   1:  PR[91,1] = PR[90,1] + 29.566;
   1:  PR[91,2] = PR[90,2] + 8.406;
   1:L PR[91] R[100]mm/sec CNT100;
   1:  PR[91,1] = PR[90,1] + 27.904;
   1:  PR[91,2] = PR[90,2] + 11.117;
   1:L PR[91] R[100]mm/sec CNT100;
   1:  PR[91,1] = PR[90,1] + 27.115;
   1:  PR[91,2] = PR[90,2] + 12.361;
   1:L PR[91] R[100]mm/sec CNT100;
   1:  PR[91,1] = PR[90,1] + 24.735;
   1:  PR[91,2] = PR[90,2] + 14.832;
   1:L PR[91] R[100]mm/sec CNT100;
   1:  PR[91,1] = PR[90,1] + 23.842;
   1:  PR[91,2] = PR[90,2] + 15.724;
   1:L PR[91] R[100]mm/sec CNT100;
   1:  PR[91,1] = PR[90,1] + 20.728;
   1:  PR[91,2] = PR[90,2] + 17.807;
   1:L PR[91] R[100]mm/sec CNT100;
   1:  PR[91,1] = PR[90,1] + 19.885;
   1:  PR[91,2] = PR[90,2] + 18.343;
   1:L PR[91] R[100]mm/sec CNT100;
   1:  PR[91,1] = PR[90,1] + 16.075;
   1:  PR[91,2] = PR[90,2] + 19.861;
   1:L PR[91] R[100]mm/sec CNT100;
   1:  PR[91,1] = PR[90,1] + 15.423;
   1:  PR[91,2] = PR[90,2] + 20.103;
   1:L PR[91] R[100]mm/sec CNT100;
   1:  PR[91,1] = PR[90,1] + 11.037;
   1:  PR[91,2] = PR[90,2] + 20.852;
   1:L PR[91] R[100]mm/sec CNT100;
   1:  PR[91,1] = PR[90,1] + 10.671;
   1:  PR[91,2] = PR[90,2] + 20.905;
   1:L PR[91] R[100]mm/sec CNT100;
   1:  PR[91,1] = PR[90,1] + 5.819;
   1:  PR[91,2] = PR[90,2] + 20.698;
   1:L PR[91] R[100]mm/sec CNT100;
   1:  PR[91,1] = PR[90,1] + 2.434;
   1:  PR[91,2] = PR[90,2] + 19.809;
   1:L PR[91] R[100]mm/sec CNT100;
   1:  PR[91,1] = PR[90,1] + 1.059;
   1:  PR[91,2] = PR[90,2] + 19.465;
   1:L PR[91] R[100]mm/sec CNT100;
   1:  PR[91,1] = PR[90,1] + 0.436;
   1:  PR[91,2] = PR[90,2] + 19.230;
   1:L PR[91] R[100]mm/sec CNT100;
   1:  PR[91] = PR[90];
   1:  PR[91,1] = PR[90,1] + -0.654;
   1:  PR[91,2] = PR[90,2] + 19.657;
   1:  PR[91,3] = PR[90,3] + 50.895;
   1:L PR[91] R[100]mm/sec CNT100;
   1:  PR[91,1] = PR[90,1] + -1.326;
   1:  PR[91,2] = PR[90,2] + 19.800;
   1:L PR[91] R[100]mm/sec CNT100;
   1:  PR[91,1] = PR[90,1] + -5.785;
   1:  PR[91,2] = PR[90,2] + 20.909;
   1:L PR[91] R[100]mm/sec CNT100;
   1:  PR[91,1] = PR[90,1] + -10.696;
   1:  PR[91,2] = PR[90,2] + 21.085;
   1:L PR[91] R[100]mm/sec CNT100;
   1:  PR[91,1] = PR[90,1] + -15.480;
   1:  PR[91,2] = PR[90,2] + 20.269;
   1:L PR[91] R[100]mm/sec CNT100;
   1:  PR[91,1] = PR[90,1] + -19.985;
   1:  PR[91,2] = PR[90,2] + 18.481;
   1:L PR[91] R[100]mm/sec CNT100;
   1:  PR[91,1] = PR[90,1] + -20.308;
   1:  PR[91,2] = PR[90,2] + 18.276;
   1:L PR[91] R[100]mm/sec CNT100;
   1:  PR[91,1] = PR[90,1] + -23.955;
   1:  PR[91,2] = PR[90,2] + 15.836;
   1:L PR[91] R[100]mm/sec CNT100;
   1:  PR[91,1] = PR[90,1] + -24.411;
   1:  PR[91,2] = PR[90,2] + 15.381;
   1:L PR[91] R[100]mm/sec CNT100;
   1:  PR[91,1] = PR[90,1] + -27.236;
   1:  PR[91,2] = PR[90,2] + 12.453;
   1:L PR[91] R[100]mm/sec CNT100;
   1:  PR[91,1] = PR[90,1] + -27.694;
   1:  PR[91,2] = PR[90,2] + 11.729;
   1:L PR[91] R[100]mm/sec CNT100;
   1:  PR[91,1] = PR[90,1] + -29.692;
   1:  PR[91,2] = PR[90,2] + 8.469;
   1:L PR[91] R[100]mm/sec CNT100;
   1:  PR[91,1] = PR[90,1] + -30.028;
   1:  PR[91,2] = PR[90,2] + 7.542;
   1:L PR[91] R[100]mm/sec CNT100;
   1:  PR[91,1] = PR[90,1] + -31.203;
   1:  PR[91,2] = PR[90,2] + 4.166;
   1:L PR[91] R[100]mm/sec CNT100;
   1:  PR[91,1] = PR[90,1] + -31.322;
   1:  PR[91,2] = PR[90,2] + 3.118;
   1:L PR[91] R[100]mm/sec CNT100;
   1:  PR[91,1] = PR[90,1] + -31.390;
   1:  PR[91,2] = PR[90,2] + 2.274;
   1:L PR[91] R[100]mm/sec CNT100;
   1:  PR[91,1] = PR[90,1] + -31.692;
   1:  PR[91,2] = PR[90,2] + -0.443;
   1:L PR[91] R[100]mm/sec CNT100;
   1:  PR[91,1] = PR[90,1] + -31.586;
   1:  PR[91,2] = PR[90,2] + -1.550;
   1:L PR[91] R[100]mm/sec CNT100;
   1:  PR[91,1] = PR[90,1] + -31.201;
   1:  PR[91,2] = PR[90,2] + -5.016;
   1:L PR[91] R[100]mm/sec CNT100;
   1:  PR[91,1] = PR[90,1] + -30.028;
   1:  PR[91,2] = PR[90,2] + -8.389;
   1:L PR[91] R[100]mm/sec CNT100;
   1:  PR[91,1] = PR[90,1] + -29.692;
   1:  PR[91,2] = PR[90,2] + -9.316;
   1:L PR[91] R[100]mm/sec CNT100;
   1:  PR[91,1] = PR[90,1] + -27.694;
   1:  PR[91,2] = PR[90,2] + -12.577;
   1:L PR[91] R[100]mm/sec CNT100;
   1:  PR[91,1] = PR[90,1] + -27.236;
   1:  PR[91,2] = PR[90,2] + -13.301;
   1:L PR[91] R[100]mm/sec CNT100;
   1:  PR[91,1] = PR[90,1] + -24.411;
   1:  PR[91,2] = PR[90,2] + -16.228;
   1:L PR[91] R[100]mm/sec CNT100;
   1:  PR[91,1] = PR[90,1] + -23.955;
   1:  PR[91,2] = PR[90,2] + -16.683;
   1:L PR[91] R[100]mm/sec CNT100;
   1:  PR[91,1] = PR[90,1] + -20.307;
   1:  PR[91,2] = PR[90,2] + -19.123;
   1:L PR[91] R[100]mm/sec CNT100;
   1:  PR[91,1] = PR[90,1] + -19.985;
   1:  PR[91,2] = PR[90,2] + -19.329;
   1:L PR[91] R[100]mm/sec CNT100;
   1:  PR[91,1] = PR[90,1] + -15.480;
   1:  PR[91,2] = PR[90,2] + -21.116;
   1:L PR[91] R[100]mm/sec CNT100;
   1:  PR[91,1] = PR[90,1] + -10.696;
   1:  PR[91,2] = PR[90,2] + -21.933;
   1:L PR[91] R[100]mm/sec CNT100;
   1:  PR[91,1] = PR[90,1] + -5.784;
   1:  PR[91,2] = PR[90,2] + -21.756;
   1:L PR[91] R[100]mm/sec CNT100;
   1:  PR[91,1] = PR[90,1] + -1.093;
   1:  PR[91,2] = PR[90,2] + -20.590;
   1:L PR[91] R[100]mm/sec CNT100;
   1:  PR[91,1] = PR[90,1] + -0.762;
   1:  PR[91,2] = PR[90,2] + -20.587;
   1:L PR[91] R[100]mm/sec CNT100;
   1:  PR[91,1] = PR[90,1] + 0.330;
   1:  PR[91,2] = PR[90,2] + -20.423;
   1:L PR[91] R[100]mm/sec CNT100;
   1:  PR[91,1] = PR[90,1] + 1.032;
   1:  PR[91,2] = PR[90,2] + -20.694;
   1:L PR[91] R[100]mm/sec CNT100;
   1:  PR[91,1] = PR[90,1] + 5.305;
   1:  PR[91,2] = PR[90,2] + -21.756;
   1:L PR[91] R[100]mm/sec CNT100;
   1:  PR[91,1] = PR[90,1] + 10.217;
   1:  PR[91,2] = PR[90,2] + -21.933;
   1:L PR[91] R[100]mm/sec CNT100;
   1:  PR[91,1] = PR[90,1] + 15.000;
   1:  PR[91,2] = PR[90,2] + -21.116;
   1:L PR[91] R[100]mm/sec CNT100;
   1:  PR[91,1] = PR[90,1] + 19.507;
   1:  PR[91,2] = PR[90,2] + -19.329;
   1:L PR[91] R[100]mm/sec CNT100;
   1:  PR[91,1] = PR[90,1] + 19.829;
   1:  PR[91,2] = PR[90,2] + -19.124;
   1:L PR[91] R[100]mm/sec CNT100;
   1:  PR[91,1] = PR[90,1] + 23.474;
   1:  PR[91,2] = PR[90,2] + -16.686;
   1:L PR[91] R[100]mm/sec CNT100;
   1:  PR[91,1] = PR[90,1] + 23.930;
   1:  PR[91,2] = PR[90,2] + -16.231;
   1:L PR[91] R[100]mm/sec CNT100;
   1:  PR[91,1] = PR[90,1] + 26.756;
   1:  PR[91,2] = PR[90,2] + -13.296;
   1:L PR[91] R[100]mm/sec CNT100;
   1:  PR[91,1] = PR[90,1] + 27.215;
   1:  PR[91,2] = PR[90,2] + -12.572;
   1:L PR[91] R[100]mm/sec CNT100;
   1:  PR[91,1] = PR[90,1] + 29.213;
   1:  PR[91,2] = PR[90,2] + -9.314;
   1:L PR[91] R[100]mm/sec CNT100;
   1:  PR[91,1] = PR[90,1] + 29.549;
   1:  PR[91,2] = PR[90,2] + -8.392;
   1:L PR[91] R[100]mm/sec CNT100;
   1:  PR[91,1] = PR[90,1] + 30.723;
   1:  PR[91,2] = PR[90,2] + -5.026;
   1:L PR[91] R[100]mm/sec CNT100;
   1:  PR[91,1] = PR[90,1] + 30.842;
   1:  PR[91,2] = PR[90,2] + -3.974;
   1:L PR[91] R[100]mm/sec CNT100;
   1:  PR[91,1] = PR[90,1] + 30.910;
   1:  PR[91,2] = PR[90,2] + -3.128;
   1:L PR[91] R[100]mm/sec CNT100;
   1:  PR[91,1] = PR[90,1] + 31.212;
   1:  PR[91,2] = PR[90,2] + -0.404;
   1:L PR[91] R[100]mm/sec CNT100;
   1:  PR[91,1] = PR[90,1] + 31.107;
   1:  PR[91,2] = PR[90,2] + 0.709;
   1:L PR[91] R[100]mm/sec CNT100;
   1:  PR[91,1] = PR[90,1] + 30.722;
   1:  PR[91,2] = PR[90,2] + 4.181;
   1:L PR[91] R[100]mm/sec CNT100;
   1:  PR[91,1] = PR[90,1] + 29.549;
   1:  PR[91,2] = PR[90,2] + 7.544;
   1:L PR[91] R[100]mm/sec CNT100;
   1:  PR[91,1] = PR[90,1] + 29.213;
   1:  PR[91,2] = PR[90,2] + 8.467;
   1:L PR[91] R[100]mm/sec CNT100;
   1:  PR[91,1] = PR[90,1] + 27.215;
   1:  PR[91,2] = PR[90,2] + 11.725;
   1:L PR[91] R[100]mm/sec CNT100;
   1:  PR[91,1] = PR[90,1] + 26.756;
   1:  PR[91,2] = PR[90,2] + 12.448;
   1:L PR[91] R[100]mm/sec CNT100;
   1:  PR[91,1] = PR[90,1] + 23.930;
   1:  PR[91,2] = PR[90,2] + 15.383;
   1:L PR[91] R[100]mm/sec CNT100;
   1:  PR[91,1] = PR[90,1] + 23.474;
   1:  PR[91,2] = PR[90,2] + 15.839;
   1:L PR[91] R[100]mm/sec CNT100;
   1:  PR[91,1] = PR[90,1] + 19.828;
   1:  PR[91,2] = PR[90,2] + 18.276;
   1:L PR[91] R[100]mm/sec CNT100;
   1:  PR[91,1] = PR[90,1] + 19.507;
   1:  PR[91,2] = PR[90,2] + 18.481;
   1:L PR[91] R[100]mm/sec CNT100;
   1:  PR[91,1] = PR[90,1] + 15.000;
   1:  PR[91,2] = PR[90,2] + 20.268;
   1:L PR[91] R[100]mm/sec CNT100;
   1:  PR[91,1] = PR[90,1] + 10.217;
   1:  PR[91,2] = PR[90,2] + 21.086;
   1:L PR[91] R[100]mm/sec CNT100;
   1:  PR[91,1] = PR[90,1] + 5.306;
   1:  PR[91,2] = PR[90,2] + 20.909;
   1:L PR[91] R[100]mm/sec CNT100;
   1:  PR[91,1] = PR[90,1] + 1.030;
   1:  PR[91,2] = PR[90,2] + 19.845;
   1:L PR[91] R[100]mm/sec CNT100;
   1:  PR[91,1] = PR[90,1] + 0.478;
   1:  PR[91,2] = PR[90,2] + 19.634;
   1:L PR[91] R[100]mm/sec CNT100;
   1:  PR[91] = PR[90];
   1:  PR[91,1] = PR[90,1] + -0.748;
   1:  PR[91,2] = PR[90,2] + 20.064;
   1:  PR[91,3] = PR[90,3] + 52.195;
   1:L PR[91] R[100]mm/sec CNT100;
   1:  PR[91,1] = PR[90,1] + -1.294;
   1:  PR[91,2] = PR[90,2] + 20.180;
   1:L PR[91] R[100]mm/sec CNT100;
   1:  PR[91,1] = PR[90,1] + -4.263;
   1:  PR[91,2] = PR[90,2] + 20.923;
   1:L PR[91] R[100]mm/sec CNT100;
   1:  PR[91,1] = PR[90,1] + -5.232;
   1:  PR[91,2] = PR[90,2] + 21.146;
   1:L PR[91] R[100]mm/sec CNT100;
   1:  PR[91,1] = PR[90,1] + -5.868;
   1:  PR[91,2] = PR[90,2] + 21.178;
   1:L PR[91] R[100]mm/sec CNT100;
   1:  PR[91,1] = PR[90,1] + -10.179;
   1:  PR[91,2] = PR[90,2] + 21.327;
   1:L PR[91] R[100]mm/sec CNT100;
   1:  PR[91,1] = PR[90,1] + -15.038;
   1:  PR[91,2] = PR[90,2] + 20.471;
   1:L PR[91] R[100]mm/sec CNT100;
   1:  PR[91,1] = PR[90,1] + -19.573;
   1:  PR[91,2] = PR[90,2] + 18.635;
   1:L PR[91] R[100]mm/sec CNT100;
   1:  PR[91,1] = PR[90,1] + -23.568;
   1:  PR[91,2] = PR[90,2] + 15.963;
   1:L PR[91] R[100]mm/sec CNT100;
   1:  PR[91,1] = PR[90,1] + -26.867;
   1:  PR[91,2] = PR[90,2] + 12.551;
   1:L PR[91] R[100]mm/sec CNT100;
   1:  PR[91,1] = PR[90,1] + -29.333;
   1:  PR[91,2] = PR[90,2] + 8.539;
   1:L PR[91] R[100]mm/sec CNT100;
   1:  PR[91,1] = PR[90,1] + -30.851;
   1:  PR[91,2] = PR[90,2] + 4.198;
   1:L PR[91] R[100]mm/sec CNT100;
   1:  PR[91,1] = PR[90,1] + -31.355;
   1:  PR[91,2] = PR[90,2] + -0.440;
   1:L PR[91] R[100]mm/sec CNT100;
   1:  PR[91,1] = PR[90,1] + -31.305;
   1:  PR[91,2] = PR[90,2] + -0.964;
   1:L PR[91] R[100]mm/sec CNT100;
   1:  PR[91,1] = PR[90,1] + -30.852;
   1:  PR[91,2] = PR[90,2] + -5.044;
   1:L PR[91] R[100]mm/sec CNT100;
   1:  PR[91,1] = PR[90,1] + -29.471;
   1:  PR[91,2] = PR[90,2] + -9.013;
   1:L PR[91] R[100]mm/sec CNT100;
   1:  PR[91,1] = PR[90,1] + -29.340;
   1:  PR[91,2] = PR[90,2] + -9.375;
   1:L PR[91] R[100]mm/sec CNT100;
   1:  PR[91,1] = PR[90,1] + -26.867;
   1:  PR[91,2] = PR[90,2] + -13.398;
   1:L PR[91] R[100]mm/sec CNT100;
   1:  PR[91,1] = PR[90,1] + -23.568;
   1:  PR[91,2] = PR[90,2] + -16.810;
   1:L PR[91] R[100]mm/sec CNT100;
   1:  PR[91,1] = PR[90,1] + -19.573;
   1:  PR[91,2] = PR[90,2] + -19.483;
   1:L PR[91] R[100]mm/sec CNT100;
   1:  PR[91,1] = PR[90,1] + -15.038;
   1:  PR[91,2] = PR[90,2] + -21.319;
   1:L PR[91] R[100]mm/sec CNT100;
   1:  PR[91,1] = PR[90,1] + -10.179;
   1:  PR[91,2] = PR[90,2] + -22.174;
   1:L PR[91] R[100]mm/sec CNT100;
   1:  PR[91,1] = PR[90,1] + -5.868;
   1:  PR[91,2] = PR[90,2] + -22.025;
   1:L PR[91] R[100]mm/sec CNT100;
   1:  PR[91,1] = PR[90,1] + -5.232;
   1:  PR[91,2] = PR[90,2] + -21.993;
   1:L PR[91] R[100]mm/sec CNT100;
   1:  PR[91,1] = PR[90,1] + -4.168;
   1:  PR[91,2] = PR[90,2] + -21.747;
   1:L PR[91] R[100]mm/sec CNT100;
   1:  PR[91,1] = PR[90,1] + -1.061;
   1:  PR[91,2] = PR[90,2] + -20.970;
   1:L PR[91] R[100]mm/sec CNT100;
   1:  PR[91,1] = PR[90,1] + -0.555;
   1:  PR[91,2] = PR[90,2] + -20.965;
   1:L PR[91] R[100]mm/sec CNT100;
   1:  PR[91,1] = PR[90,1] + 0.380;
   1:  PR[91,2] = PR[90,2] + -20.825;
   1:L PR[91] R[100]mm/sec CNT100;
   1:  PR[91,1] = PR[90,1] + 1.014;
   1:  PR[91,2] = PR[90,2] + -21.078;
   1:L PR[91] R[100]mm/sec CNT100;
   1:  PR[91,1] = PR[90,1] + 3.691;
   1:  PR[91,2] = PR[90,2] + -21.747;
   1:L PR[91] R[100]mm/sec CNT100;
   1:  PR[91,1] = PR[90,1] + 4.754;
   1:  PR[91,2] = PR[90,2] + -21.994;
   1:L PR[91] R[100]mm/sec CNT100;
   1:  PR[91,1] = PR[90,1] + 5.389;
   1:  PR[91,2] = PR[90,2] + -22.025;
   1:L PR[91] R[100]mm/sec CNT100;
   1:  PR[91,1] = PR[90,1] + 9.700;
   1:  PR[91,2] = PR[90,2] + -22.175;
   1:L PR[91] R[100]mm/sec CNT100;
   1:  PR[91,1] = PR[90,1] + 14.559;
   1:  PR[91,2] = PR[90,2] + -21.318;
   1:L PR[91] R[100]mm/sec CNT100;
   1:  PR[91,1] = PR[90,1] + 19.094;
   1:  PR[91,2] = PR[90,2] + -19.483;
   1:L PR[91] R[100]mm/sec CNT100;
   1:  PR[91,1] = PR[90,1] + 23.087;
   1:  PR[91,2] = PR[90,2] + -16.812;
   1:L PR[91] R[100]mm/sec CNT100;
   1:  PR[91,1] = PR[90,1] + 26.398;
   1:  PR[91,2] = PR[90,2] + -13.382;
   1:L PR[91] R[100]mm/sec CNT100;
   1:  PR[91,1] = PR[90,1] + 26.526;
   1:  PR[91,2] = PR[90,2] + -13.180;
   1:L PR[91] R[100]mm/sec CNT100;
   1:  PR[91,1] = PR[90,1] + 28.853;
   1:  PR[91,2] = PR[90,2] + -9.387;
   1:L PR[91] R[100]mm/sec CNT100;
   1:  PR[91,1] = PR[90,1] + 30.371;
   1:  PR[91,2] = PR[90,2] + -5.056;
   1:L PR[91] R[100]mm/sec CNT100;
   1:  PR[91,1] = PR[90,1] + 30.875;
   1:  PR[91,2] = PR[90,2] + -0.407;
   1:L PR[91] R[100]mm/sec CNT100;
   1:  PR[91,1] = PR[90,1] + 30.825;
   1:  PR[91,2] = PR[90,2] + 0.121;
   1:L PR[91] R[100]mm/sec CNT100;
   1:  PR[91,1] = PR[90,1] + 30.372;
   1:  PR[91,2] = PR[90,2] + 4.206;
   1:L PR[91] R[100]mm/sec CNT100;
   1:  PR[91,1] = PR[90,1] + 28.854;
   1:  PR[91,2] = PR[90,2] + 8.538;
   1:L PR[91] R[100]mm/sec CNT100;
   1:  PR[91,1] = PR[90,1] + 26.386;
   1:  PR[91,2] = PR[90,2] + 12.548;
   1:L PR[91] R[100]mm/sec CNT100;
   1:  PR[91,1] = PR[90,1] + 23.125;
   1:  PR[91,2] = PR[90,2] + 15.934;
   1:L PR[91] R[100]mm/sec CNT100;
   1:  PR[91,1] = PR[90,1] + 23.106;
   1:  PR[91,2] = PR[90,2] + 15.953;
   1:L PR[91] R[100]mm/sec CNT100;
   1:  PR[91,1] = PR[90,1] + 19.094;
   1:  PR[91,2] = PR[90,2] + 18.635;
   1:L PR[91] R[100]mm/sec CNT100;
   1:  PR[91,1] = PR[90,1] + 14.558;
   1:  PR[91,2] = PR[90,2] + 20.471;
   1:L PR[91] R[100]mm/sec CNT100;
   1:  PR[91,1] = PR[90,1] + 9.699;
   1:  PR[91,2] = PR[90,2] + 21.327;
   1:L PR[91] R[100]mm/sec CNT100;
   1:  PR[91,1] = PR[90,1] + 5.388;
   1:  PR[91,2] = PR[90,2] + 21.178;
   1:L PR[91] R[100]mm/sec CNT100;
   1:  PR[91,1] = PR[90,1] + 4.753;
   1:  PR[91,2] = PR[90,2] + 21.146;
   1:L PR[91] R[100]mm/sec CNT100;
   1:  PR[91,1] = PR[90,1] + 3.785;
   1:  PR[91,2] = PR[90,2] + 20.923;
   1:L PR[91] R[100]mm/sec CNT100;
   1:  PR[91,1] = PR[90,1] + 1.008;
   1:  PR[91,2] = PR[90,2] + 20.228;
   1:L PR[91] R[100]mm/sec CNT100;
   1:  PR[91,1] = PR[90,1] + 0.523;
   1:  PR[91,2] = PR[90,2] + 20.038;
   1:L PR[91] R[100]mm/sec CNT100;
   1:  PR[91] = PR[90];
   1:  PR[91,1] = PR[90,1] + -0.881;
   1:  PR[91,2] = PR[90,2] + 20.471;
   1:  PR[91,3] = PR[90,3] + 53.495;
   1:L PR[91] R[100]mm/sec CNT100;
   1:  PR[91,1] = PR[90,1] + -2.896;
   1:  PR[91,2] = PR[90,2] + 20.968;
   1:L PR[91] R[100]mm/sec CNT100;
   1:  PR[91,1] = PR[90,1] + -4.684;
   1:  PR[91,2] = PR[90,2] + 21.381;
   1:L PR[91] R[100]mm/sec CNT100;
   1:  PR[91,1] = PR[90,1] + -5.909;
   1:  PR[91,2] = PR[90,2] + 21.442;
   1:L PR[91] R[100]mm/sec CNT100;
   1:  PR[91,1] = PR[90,1] + -9.679;
   1:  PR[91,2] = PR[90,2] + 21.572;
   1:L PR[91] R[100]mm/sec CNT100;
   1:  PR[91,1] = PR[90,1] + -10.612;
   1:  PR[91,2] = PR[90,2] + 21.419;
   1:L PR[91] R[100]mm/sec CNT100;
   1:  PR[91,1] = PR[90,1] + -14.569;
   1:  PR[91,2] = PR[90,2] + 20.717;
   1:L PR[91] R[100]mm/sec CNT100;
   1:  PR[91,1] = PR[90,1] + -19.147;
   1:  PR[91,2] = PR[90,2] + 18.866;
   1:L PR[91] R[100]mm/sec CNT100;
   1:  PR[91,1] = PR[90,1] + -23.184;
   1:  PR[91,2] = PR[90,2] + 16.135;
   1:L PR[91] R[100]mm/sec CNT100;
   1:  PR[91,1] = PR[90,1] + -26.505;
   1:  PR[91,2] = PR[90,2] + 12.662;
   1:L PR[91] R[100]mm/sec CNT100;
   1:  PR[91,1] = PR[90,1] + -28.978;
   1:  PR[91,2] = PR[90,2] + 8.605;
   1:L PR[91] R[100]mm/sec CNT100;
   1:  PR[91,1] = PR[90,1] + -30.503;
   1:  PR[91,2] = PR[90,2] + 4.226;
   1:L PR[91] R[100]mm/sec CNT100;
   1:  PR[91,1] = PR[90,1] + -31.016;
   1:  PR[91,2] = PR[90,2] + -0.424;
   1:L PR[91] R[100]mm/sec CNT100;
   1:  PR[91,1] = PR[90,1] + -30.503;
   1:  PR[91,2] = PR[90,2] + -5.073;
   1:L PR[91] R[100]mm/sec CNT100;
   1:  PR[91,1] = PR[90,1] + -28.978;
   1:  PR[91,2] = PR[90,2] + -9.453;
   1:L PR[91] R[100]mm/sec CNT100;
   1:  PR[91,1] = PR[90,1] + -26.504;
   1:  PR[91,2] = PR[90,2] + -13.510;
   1:L PR[91] R[100]mm/sec CNT100;
   1:  PR[91,1] = PR[90,1] + -23.184;
   1:  PR[91,2] = PR[90,2] + -16.982;
   1:L PR[91] R[100]mm/sec CNT100;
   1:  PR[91,1] = PR[90,1] + -19.147;
   1:  PR[91,2] = PR[90,2] + -19.713;
   1:L PR[91] R[100]mm/sec CNT100;
   1:  PR[91,1] = PR[90,1] + -14.569;
   1:  PR[91,2] = PR[90,2] + -21.564;
   1:L PR[91] R[100]mm/sec CNT100;
   1:  PR[91,1] = PR[90,1] + -10.613;
   1:  PR[91,2] = PR[90,2] + -22.266;
   1:L PR[91] R[100]mm/sec CNT100;
   1:  PR[91,1] = PR[90,1] + -9.680;
   1:  PR[91,2] = PR[90,2] + -22.420;
   1:L PR[91] R[100]mm/sec CNT100;
   1:  PR[91,1] = PR[90,1] + -5.909;
   1:  PR[91,2] = PR[90,2] + -22.289;
   1:L PR[91] R[100]mm/sec CNT100;
   1:  PR[91,1] = PR[90,1] + -4.684;
   1:  PR[91,2] = PR[90,2] + -22.228;
   1:L PR[91] R[100]mm/sec CNT100;
   1:  PR[91,1] = PR[90,1] + -2.741;
   1:  PR[91,2] = PR[90,2] + -21.778;
   1:L PR[91] R[100]mm/sec CNT100;
   1:  PR[91,1] = PR[90,1] + -1.027;
   1:  PR[91,2] = PR[90,2] + -21.350;
   1:L PR[91] R[100]mm/sec CNT100;
   1:  PR[91,1] = PR[90,1] + -0.348;
   1:  PR[91,2] = PR[90,2] + -21.343;
   1:L PR[91] R[100]mm/sec CNT100;
   1:  PR[91,1] = PR[90,1] + 0.447;
   1:  PR[91,2] = PR[90,2] + -21.224;
   1:L PR[91] R[100]mm/sec CNT100;
   1:  PR[91,1] = PR[90,1] + 1.010;
   1:  PR[91,2] = PR[90,2] + -21.465;
   1:L PR[91] R[100]mm/sec CNT100;
   1:  PR[91,1] = PR[90,1] + 2.263;
   1:  PR[91,2] = PR[90,2] + -21.778;
   1:L PR[91] R[100]mm/sec CNT100;
   1:  PR[91,1] = PR[90,1] + 4.205;
   1:  PR[91,2] = PR[90,2] + -22.228;
   1:L PR[91] R[100]mm/sec CNT100;
   1:  PR[91,1] = PR[90,1] + 5.430;
   1:  PR[91,2] = PR[90,2] + -22.289;
   1:L PR[91] R[100]mm/sec CNT100;
   1:  PR[91,1] = PR[90,1] + 9.201;
   1:  PR[91,2] = PR[90,2] + -22.420;
   1:L PR[91] R[100]mm/sec CNT100;
   1:  PR[91,1] = PR[90,1] + 10.133;
   1:  PR[91,2] = PR[90,2] + -22.266;
   1:L PR[91] R[100]mm/sec CNT100;
   1:  PR[91,1] = PR[90,1] + 14.090;
   1:  PR[91,2] = PR[90,2] + -21.563;
   1:L PR[91] R[100]mm/sec CNT100;
   1:  PR[91,1] = PR[90,1] + 18.672;
   1:  PR[91,2] = PR[90,2] + -19.712;
   1:L PR[91] R[100]mm/sec CNT100;
   1:  PR[91,1] = PR[90,1] + 18.975;
   1:  PR[91,2] = PR[90,2] + -19.508;
   1:L PR[91] R[100]mm/sec CNT100;
   1:  PR[91,1] = PR[90,1] + 22.704;
   1:  PR[91,2] = PR[90,2] + -16.984;
   1:L PR[91] R[100]mm/sec CNT100;
   1:  PR[91,1] = PR[90,1] + 26.025;
   1:  PR[91,2] = PR[90,2] + -13.505;
   1:L PR[91] R[100]mm/sec CNT100;
   1:  PR[91,1] = PR[90,1] + 28.499;
   1:  PR[91,2] = PR[90,2] + -9.451;
   1:L PR[91] R[100]mm/sec CNT100;
   1:  PR[91,1] = PR[90,1] + 30.023;
   1:  PR[91,2] = PR[90,2] + -5.083;
   1:L PR[91] R[100]mm/sec CNT100;
   1:  PR[91,1] = PR[90,1] + 30.536;
   1:  PR[91,2] = PR[90,2] + -0.424;
   1:L PR[91] R[100]mm/sec CNT100;
   1:  PR[91,1] = PR[90,1] + 30.023;
   1:  PR[91,2] = PR[90,2] + 4.236;
   1:L PR[91] R[100]mm/sec CNT100;
   1:  PR[91,1] = PR[90,1] + 28.499;
   1:  PR[91,2] = PR[90,2] + 8.604;
   1:L PR[91] R[100]mm/sec CNT100;
   1:  PR[91,1] = PR[90,1] + 26.025;
   1:  PR[91,2] = PR[90,2] + 12.658;
   1:L PR[91] R[100]mm/sec CNT100;
   1:  PR[91,1] = PR[90,1] + 22.704;
   1:  PR[91,2] = PR[90,2] + 16.137;
   1:L PR[91] R[100]mm/sec CNT100;
   1:  PR[91,1] = PR[90,1] + 18.668;
   1:  PR[91,2] = PR[90,2] + 18.866;
   1:L PR[91] R[100]mm/sec CNT100;
   1:  PR[91,1] = PR[90,1] + 14.090;
   1:  PR[91,2] = PR[90,2] + 20.716;
   1:L PR[91] R[100]mm/sec CNT100;
   1:  PR[91,1] = PR[90,1] + 10.133;
   1:  PR[91,2] = PR[90,2] + 21.419;
   1:L PR[91] R[100]mm/sec CNT100;
   1:  PR[91,1] = PR[90,1] + 9.200;
   1:  PR[91,2] = PR[90,2] + 21.573;
   1:L PR[91] R[100]mm/sec CNT100;
   1:  PR[91,1] = PR[90,1] + 5.429;
   1:  PR[91,2] = PR[90,2] + 21.442;
   1:L PR[91] R[100]mm/sec CNT100;
   1:  PR[91,1] = PR[90,1] + 4.205;
   1:  PR[91,2] = PR[90,2] + 21.381;
   1:L PR[91] R[100]mm/sec CNT100;
   1:  PR[91,1] = PR[90,1] + 2.422;
   1:  PR[91,2] = PR[90,2] + 20.969;
   1:L PR[91] R[100]mm/sec CNT100;
   1:  PR[91,1] = PR[90,1] + 0.996;
   1:  PR[91,2] = PR[90,2] + 20.612;
   1:L PR[91] R[100]mm/sec CNT100;
   1:  PR[91,1] = PR[90,1] + 0.581;
   1:  PR[91,2] = PR[90,2] + 20.441;
   1:L PR[91] R[100]mm/sec CNT100;
   1:  PR[91] = PR[90];
   1:  PR[91,1] = PR[90,1] + -0.957;
   1:  PR[91,2] = PR[90,2] + 20.877;
   1:  PR[91,3] = PR[90,3] + 54.795;
   1:L PR[91] R[100]mm/sec CNT100;
   1:  PR[91,1] = PR[90,1] + -4.137;
   1:  PR[91,2] = PR[90,2] + 21.616;
   1:L PR[91] R[100]mm/sec CNT100;
   1:  PR[91,1] = PR[90,1] + -5.949;
   1:  PR[91,2] = PR[90,2] + 21.706;
   1:L PR[91] R[100]mm/sec CNT100;
   1:  PR[91,1] = PR[90,1] + -9.166;
   1:  PR[91,2] = PR[90,2] + 21.817;
   1:L PR[91] R[100]mm/sec CNT100;
   1:  PR[91,1] = PR[90,1] + -10.703;
   1:  PR[91,2] = PR[90,2] + 21.565;
   1:L PR[91] R[100]mm/sec CNT100;
   1:  PR[91,1] = PR[90,1] + -14.103;
   1:  PR[91,2] = PR[90,2] + 20.961;
   1:L PR[91] R[100]mm/sec CNT100;
   1:  PR[91,1] = PR[90,1] + -18.727;
   1:  PR[91,2] = PR[90,2] + 19.097;
   1:L PR[91] R[100]mm/sec CNT100;
   1:  PR[91,1] = PR[90,1] + -22.806;
   1:  PR[91,2] = PR[90,2] + 16.340;
   1:L PR[91] R[100]mm/sec CNT100;
   1:  PR[91,1] = PR[90,1] + -26.163;
   1:  PR[91,2] = PR[90,2] + 12.830;
   1:L PR[91] R[100]mm/sec CNT100;
   1:  PR[91,1] = PR[90,1] + -28.661;
   1:  PR[91,2] = PR[90,2] + 8.724;
   1:L PR[91] R[100]mm/sec CNT100;
   1:  PR[91,1] = PR[90,1] + -30.195;
   1:  PR[91,2] = PR[90,2] + 4.282;
   1:L PR[91] R[100]mm/sec CNT100;
   1:  PR[91,1] = PR[90,1] + -30.706;
   1:  PR[91,2] = PR[90,2] + -0.422;
   1:L PR[91] R[100]mm/sec CNT100;
   1:  PR[91,1] = PR[90,1] + -30.235;
   1:  PR[91,2] = PR[90,2] + -4.708;
   1:L PR[91] R[100]mm/sec CNT100;
   1:  PR[91,1] = PR[90,1] + -30.219;
   1:  PR[91,2] = PR[90,2] + -4.916;
   1:L PR[91] R[100]mm/sec CNT100;
   1:  PR[91,1] = PR[90,1] + -30.196;
   1:  PR[91,2] = PR[90,2] + -5.127;
   1:L PR[91] R[100]mm/sec CNT100;
   1:  PR[91,1] = PR[90,1] + -28.661;
   1:  PR[91,2] = PR[90,2] + -9.571;
   1:L PR[91] R[100]mm/sec CNT100;
   1:  PR[91,1] = PR[90,1] + -26.163;
   1:  PR[91,2] = PR[90,2] + -13.677;
   1:L PR[91] R[100]mm/sec CNT100;
   1:  PR[91,1] = PR[90,1] + -22.807;
   1:  PR[91,2] = PR[90,2] + -17.187;
   1:L PR[91] R[100]mm/sec CNT100;
   1:  PR[91,1] = PR[90,1] + -18.727;
   1:  PR[91,2] = PR[90,2] + -19.944;
   1:L PR[91] R[100]mm/sec CNT100;
   1:  PR[91,1] = PR[90,1] + -14.103;
   1:  PR[91,2] = PR[90,2] + -21.808;
   1:L PR[91] R[100]mm/sec CNT100;
   1:  PR[91,1] = PR[90,1] + -10.705;
   1:  PR[91,2] = PR[90,2] + -22.411;
   1:L PR[91] R[100]mm/sec CNT100;
   1:  PR[91,1] = PR[90,1] + -9.167;
   1:  PR[91,2] = PR[90,2] + -22.664;
   1:L PR[91] R[100]mm/sec CNT100;
   1:  PR[91,1] = PR[90,1] + -5.950;
   1:  PR[91,2] = PR[90,2] + -22.553;
   1:L PR[91] R[100]mm/sec CNT100;
   1:  PR[91,1] = PR[90,1] + -4.135;
   1:  PR[91,2] = PR[90,2] + -22.462;
   1:L PR[91] R[100]mm/sec CNT100;
   1:  PR[91,1] = PR[90,1] + -0.972;
   1:  PR[91,2] = PR[90,2] + -21.729;
   1:L PR[91] R[100]mm/sec CNT100;
   1:  PR[91,1] = PR[90,1] + -0.140;
   1:  PR[91,2] = PR[90,2] + -21.721;
   1:L PR[91] R[100]mm/sec CNT100;
   1:  PR[91,1] = PR[90,1] + 0.624;
   1:  PR[91,2] = PR[90,2] + -21.607;
   1:L PR[91] R[100]mm/sec CNT100;
   1:  PR[91,1] = PR[90,1] + 1.092;
   1:  PR[91,2] = PR[90,2] + -21.870;
   1:L PR[91] R[100]mm/sec CNT100;
   1:  PR[91,1] = PR[90,1] + 1.544;
   1:  PR[91,2] = PR[90,2] + -21.979;
   1:L PR[91] R[100]mm/sec CNT100;
   1:  PR[91,1] = PR[90,1] + 3.653;
   1:  PR[91,2] = PR[90,2] + -22.462;
   1:L PR[91] R[100]mm/sec CNT100;
   1:  PR[91,1] = PR[90,1] + 5.471;
   1:  PR[91,2] = PR[90,2] + -22.553;
   1:L PR[91] R[100]mm/sec CNT100;
   1:  PR[91,1] = PR[90,1] + 8.688;
   1:  PR[91,2] = PR[90,2] + -22.665;
   1:L PR[91] R[100]mm/sec CNT100;
   1:  PR[91,1] = PR[90,1] + 10.225;
   1:  PR[91,2] = PR[90,2] + -22.412;
   1:L PR[91] R[100]mm/sec CNT100;
   1:  PR[91,1] = PR[90,1] + 13.624;
   1:  PR[91,2] = PR[90,2] + -21.807;
   1:L PR[91] R[100]mm/sec CNT100;
   1:  PR[91,1] = PR[90,1] + 18.249;
   1:  PR[91,2] = PR[90,2] + -19.944;
   1:L PR[91] R[100]mm/sec CNT100;
   1:  PR[91,1] = PR[90,1] + 22.326;
   1:  PR[91,2] = PR[90,2] + -17.189;
   1:L PR[91] R[100]mm/sec CNT100;
   1:  PR[91,1] = PR[90,1] + 25.684;
   1:  PR[91,2] = PR[90,2] + -13.673;
   1:L PR[91] R[100]mm/sec CNT100;
   1:  PR[91,1] = PR[90,1] + 28.182;
   1:  PR[91,2] = PR[90,2] + -9.570;
   1:L PR[91] R[100]mm/sec CNT100;
   1:  PR[91,1] = PR[90,1] + 29.715;
   1:  PR[91,2] = PR[90,2] + -5.138;
   1:L PR[91] R[100]mm/sec CNT100;
   1:  PR[91,1] = PR[90,1] + 30.227;
   1:  PR[91,2] = PR[90,2] + -0.424;
   1:L PR[91] R[100]mm/sec CNT100;
   1:  PR[91,1] = PR[90,1] + 29.715;
   1:  PR[91,2] = PR[90,2] + 4.291;
   1:L PR[91] R[100]mm/sec CNT100;
   1:  PR[91,1] = PR[90,1] + 28.182;
   1:  PR[91,2] = PR[90,2] + 8.723;
   1:L PR[91] R[100]mm/sec CNT100;
   1:  PR[91,1] = PR[90,1] + 25.683;
   1:  PR[91,2] = PR[90,2] + 12.826;
   1:L PR[91] R[100]mm/sec CNT100;
   1:  PR[91,1] = PR[90,1] + 22.326;
   1:  PR[91,2] = PR[90,2] + 16.342;
   1:L PR[91] R[100]mm/sec CNT100;
   1:  PR[91,1] = PR[90,1] + 18.248;
   1:  PR[91,2] = PR[90,2] + 19.097;
   1:L PR[91] R[100]mm/sec CNT100;
   1:  PR[91,1] = PR[90,1] + 13.623;
   1:  PR[91,2] = PR[90,2] + 20.960;
   1:L PR[91] R[100]mm/sec CNT100;
   1:  PR[91,1] = PR[90,1] + 10.224;
   1:  PR[91,2] = PR[90,2] + 21.565;
   1:L PR[91] R[100]mm/sec CNT100;
   1:  PR[91,1] = PR[90,1] + 8.686;
   1:  PR[91,2] = PR[90,2] + 21.817;
   1:L PR[91] R[100]mm/sec CNT100;
   1:  PR[91,1] = PR[90,1] + 5.470;
   1:  PR[91,2] = PR[90,2] + 21.706;
   1:L PR[91] R[100]mm/sec CNT100;
   1:  PR[91,1] = PR[90,1] + 3.654;
   1:  PR[91,2] = PR[90,2] + 21.615;
   1:L PR[91] R[100]mm/sec CNT100;
   1:  PR[91,1] = PR[90,1] + 1.554;
   1:  PR[91,2] = PR[90,2] + 21.134;
   1:L PR[91] R[100]mm/sec CNT100;
   1:  PR[91,1] = PR[90,1] + 1.039;
   1:  PR[91,2] = PR[90,2] + 21.009;
   1:L PR[91] R[100]mm/sec CNT100;
   1:  PR[91,1] = PR[90,1] + 0.705;
   1:  PR[91,2] = PR[90,2] + 20.843;
   1:L PR[91] R[100]mm/sec CNT100;
   1:  PR[91] = PR[90];
   1:  PR[91,1] = PR[90,1] + -0.921;
   1:  PR[91,2] = PR[90,2] + 21.235;
   1:  PR[91,3] = PR[90,3] + 56.095;
   1:L PR[91] R[100]mm/sec CNT100;
   1:  PR[91,1] = PR[90,1] + -3.587;
   1:  PR[91,2] = PR[90,2] + 21.850;
   1:L PR[91] R[100]mm/sec CNT100;
   1:  PR[91,1] = PR[90,1] + -5.989;
   1:  PR[91,2] = PR[90,2] + 21.970;
   1:L PR[91] R[100]mm/sec CNT100;
   1:  PR[91,1] = PR[90,1] + -8.652;
   1:  PR[91,2] = PR[90,2] + 22.062;
   1:L PR[91] R[100]mm/sec CNT100;
   1:  PR[91,1] = PR[90,1] + -10.795;
   1:  PR[91,2] = PR[90,2] + 21.710;
   1:L PR[91] R[100]mm/sec CNT100;
   1:  PR[91,1] = PR[90,1] + -13.642;
   1:  PR[91,2] = PR[90,2] + 21.204;
   1:L PR[91] R[100]mm/sec CNT100;
   1:  PR[91,1] = PR[90,1] + -15.420;
   1:  PR[91,2] = PR[90,2] + 20.500;
   1:L PR[91] R[100]mm/sec CNT100;
   1:  PR[91,1] = PR[90,1] + -18.303;
   1:  PR[91,2] = PR[90,2] + 19.330;
   1:L PR[91] R[100]mm/sec CNT100;
   1:  PR[91,1] = PR[90,1] + -22.428;
   1:  PR[91,2] = PR[90,2] + 16.545;
   1:L PR[91] R[100]mm/sec CNT100;
   1:  PR[91,1] = PR[90,1] + -25.823;
   1:  PR[91,2] = PR[90,2] + 12.997;
   1:L PR[91] R[100]mm/sec CNT100;
   1:  PR[91,1] = PR[90,1] + -28.350;
   1:  PR[91,2] = PR[90,2] + 8.843;
   1:L PR[91] R[100]mm/sec CNT100;
   1:  PR[91,1] = PR[90,1] + -29.903;
   1:  PR[91,2] = PR[90,2] + 4.339;
   1:L PR[91] R[100]mm/sec CNT100;
   1:  PR[91,1] = PR[90,1] + -30.326;
   1:  PR[91,2] = PR[90,2] + 0.489;
   1:L PR[91] R[100]mm/sec CNT100;
   1:  PR[91,1] = PR[90,1] + -30.412;
   1:  PR[91,2] = PR[90,2] + -0.407;
   1:L PR[91] R[100]mm/sec CNT100;
   1:  PR[91,1] = PR[90,1] + -30.038;
   1:  PR[91,2] = PR[90,2] + -3.805;
   1:L PR[91] R[100]mm/sec CNT100;
   1:  PR[91,1] = PR[90,1] + -30.002;
   1:  PR[91,2] = PR[90,2] + -4.289;
   1:L PR[91] R[100]mm/sec CNT100;
   1:  PR[91,1] = PR[90,1] + -29.903;
   1:  PR[91,2] = PR[90,2] + -5.186;
   1:L PR[91] R[100]mm/sec CNT100;
   1:  PR[91,1] = PR[90,1] + -28.350;
   1:  PR[91,2] = PR[90,2] + -9.690;
   1:L PR[91] R[100]mm/sec CNT100;
   1:  PR[91,1] = PR[90,1] + -25.823;
   1:  PR[91,2] = PR[90,2] + -13.844;
   1:L PR[91] R[100]mm/sec CNT100;
   1:  PR[91,1] = PR[90,1] + -22.429;
   1:  PR[91,2] = PR[90,2] + -17.392;
   1:L PR[91] R[100]mm/sec CNT100;
   1:  PR[91,1] = PR[90,1] + -18.304;
   1:  PR[91,2] = PR[90,2] + -20.177;
   1:L PR[91] R[100]mm/sec CNT100;
   1:  PR[91,1] = PR[90,1] + -15.421;
   1:  PR[91,2] = PR[90,2] + -21.347;
   1:L PR[91] R[100]mm/sec CNT100;
   1:  PR[91,1] = PR[90,1] + -13.643;
   1:  PR[91,2] = PR[90,2] + -22.051;
   1:L PR[91] R[100]mm/sec CNT100;
   1:  PR[91,1] = PR[90,1] + -10.797;
   1:  PR[91,2] = PR[90,2] + -22.557;
   1:L PR[91] R[100]mm/sec CNT100;
   1:  PR[91,1] = PR[90,1] + -8.653;
   1:  PR[91,2] = PR[90,2] + -22.909;
   1:L PR[91] R[100]mm/sec CNT100;
   1:  PR[91,1] = PR[90,1] + -5.991;
   1:  PR[91,2] = PR[90,2] + -22.817;
   1:L PR[91] R[100]mm/sec CNT100;
   1:  PR[91,1] = PR[90,1] + -3.586;
   1:  PR[91,2] = PR[90,2] + -22.697;
   1:L PR[91] R[100]mm/sec CNT100;
   1:  PR[91,1] = PR[90,1] + -0.919;
   1:  PR[91,2] = PR[90,2] + -22.080;
   1:L PR[91] R[100]mm/sec CNT100;
   1:  PR[91,1] = PR[90,1] + 0.457;
   1:  PR[91,2] = PR[90,2] + -22.091;
   1:L PR[91] R[100]mm/sec CNT100;
   1:  PR[91,1] = PR[90,1] + 3.104;
   1:  PR[91,2] = PR[90,2] + -22.697;
   1:L PR[91] R[100]mm/sec CNT100;
   1:  PR[91,1] = PR[90,1] + 5.512;
   1:  PR[91,2] = PR[90,2] + -22.817;
   1:L PR[91] R[100]mm/sec CNT100;
   1:  PR[91,1] = PR[90,1] + 8.175;
   1:  PR[91,2] = PR[90,2] + -22.909;
   1:L PR[91] R[100]mm/sec CNT100;
   1:  PR[91,1] = PR[90,1] + 10.317;
   1:  PR[91,2] = PR[90,2] + -22.557;
   1:L PR[91] R[100]mm/sec CNT100;
   1:  PR[91,1] = PR[90,1] + 13.164;
   1:  PR[91,2] = PR[90,2] + -22.051;
   1:L PR[91] R[100]mm/sec CNT100;
   1:  PR[91,1] = PR[90,1] + 14.942;
   1:  PR[91,2] = PR[90,2] + -21.346;
   1:L PR[91] R[100]mm/sec CNT100;
   1:  PR[91,1] = PR[90,1] + 17.825;
   1:  PR[91,2] = PR[90,2] + -20.177;
   1:L PR[91] R[100]mm/sec CNT100;
   1:  PR[91,1] = PR[90,1] + 21.949;
   1:  PR[91,2] = PR[90,2] + -17.393;
   1:L PR[91] R[100]mm/sec CNT100;
   1:  PR[91,1] = PR[90,1] + 25.343;
   1:  PR[91,2] = PR[90,2] + -13.840;
   1:L PR[91] R[100]mm/sec CNT100;
   1:  PR[91,1] = PR[90,1] + 27.871;
   1:  PR[91,2] = PR[90,2] + -9.689;
   1:L PR[91] R[100]mm/sec CNT100;
   1:  PR[91,1] = PR[90,1] + 29.423;
   1:  PR[91,2] = PR[90,2] + -5.195;
   1:L PR[91] R[100]mm/sec CNT100;
   1:  PR[91,1] = PR[90,1] + 29.847;
   1:  PR[91,2] = PR[90,2] + -1.337;
   1:L PR[91] R[100]mm/sec CNT100;
   1:  PR[91,1] = PR[90,1] + 29.933;
   1:  PR[91,2] = PR[90,2] + -0.440;
   1:L PR[91] R[100]mm/sec CNT100;
   1:  PR[91,1] = PR[90,1] + 29.558;
   1:  PR[91,2] = PR[90,2] + 2.965;
   1:L PR[91] R[100]mm/sec CNT100;
   1:  PR[91,1] = PR[90,1] + 29.522;
   1:  PR[91,2] = PR[90,2] + 3.450;
   1:L PR[91] R[100]mm/sec CNT100;
   1:  PR[91,1] = PR[90,1] + 29.423;
   1:  PR[91,2] = PR[90,2] + 4.347;
   1:L PR[91] R[100]mm/sec CNT100;
   1:  PR[91,1] = PR[90,1] + 27.871;
   1:  PR[91,2] = PR[90,2] + 8.842;
   1:L PR[91] R[100]mm/sec CNT100;
   1:  PR[91,1] = PR[90,1] + 25.343;
   1:  PR[91,2] = PR[90,2] + 12.993;
   1:L PR[91] R[100]mm/sec CNT100;
   1:  PR[91,1] = PR[90,1] + 21.948;
   1:  PR[91,2] = PR[90,2] + 16.547;
   1:L PR[91] R[100]mm/sec CNT100;
   1:  PR[91,1] = PR[90,1] + 17.825;
   1:  PR[91,2] = PR[90,2] + 19.330;
   1:L PR[91] R[100]mm/sec CNT100;
   1:  PR[91,1] = PR[90,1] + 14.941;
   1:  PR[91,2] = PR[90,2] + 20.500;
   1:L PR[91] R[100]mm/sec CNT100;
   1:  PR[91,1] = PR[90,1] + 13.163;
   1:  PR[91,2] = PR[90,2] + 21.204;
   1:L PR[91] R[100]mm/sec CNT100;
   1:  PR[91,1] = PR[90,1] + 10.316;
   1:  PR[91,2] = PR[90,2] + 21.710;
   1:L PR[91] R[100]mm/sec CNT100;
   1:  PR[91,1] = PR[90,1] + 8.173;
   1:  PR[91,2] = PR[90,2] + 22.062;
   1:L PR[91] R[100]mm/sec CNT100;
   1:  PR[91,1] = PR[90,1] + 5.511;
   1:  PR[91,2] = PR[90,2] + 21.970;
   1:L PR[91] R[100]mm/sec CNT100;
   1:  PR[91,1] = PR[90,1] + 3.106;
   1:  PR[91,2] = PR[90,2] + 21.850;
   1:L PR[91] R[100]mm/sec CNT100;
   1:  PR[91,1] = PR[90,1] + 0.455;
   1:  PR[91,2] = PR[90,2] + 21.243;
   1:L PR[91] R[100]mm/sec CNT100;
   1:  PR[91] = PR[90];
   1:  PR[91,1] = PR[90,1] + -0.891;
   1:  PR[91,2] = PR[90,2] + 21.589;
   1:  PR[91,3] = PR[90,3] + 57.395;
   1:L PR[91] R[100]mm/sec CNT100;
   1:  PR[91,1] = PR[90,1] + -3.039;
   1:  PR[91,2] = PR[90,2] + 22.085;
   1:L PR[91] R[100]mm/sec CNT100;
   1:  PR[91,1] = PR[90,1] + -6.030;
   1:  PR[91,2] = PR[90,2] + 22.234;
   1:L PR[91] R[100]mm/sec CNT100;
   1:  PR[91,1] = PR[90,1] + -8.139;
   1:  PR[91,2] = PR[90,2] + 22.307;
   1:L PR[91] R[100]mm/sec CNT100;
   1:  PR[91,1] = PR[90,1] + -10.887;
   1:  PR[91,2] = PR[90,2] + 21.855;
   1:L PR[91] R[100]mm/sec CNT100;
   1:  PR[91,1] = PR[90,1] + -13.175;
   1:  PR[91,2] = PR[90,2] + 21.449;
   1:L PR[91] R[100]mm/sec CNT100;
   1:  PR[91,1] = PR[90,1] + -15.538;
   1:  PR[91,2] = PR[90,2] + 20.513;
   1:L PR[91] R[100]mm/sec CNT100;
   1:  PR[91,1] = PR[90,1] + -17.882;
   1:  PR[91,2] = PR[90,2] + 19.562;
   1:L PR[91] R[100]mm/sec CNT100;
   1:  PR[91,1] = PR[90,1] + -22.051;
   1:  PR[91,2] = PR[90,2] + 16.750;
   1:L PR[91] R[100]mm/sec CNT100;
   1:  PR[91,1] = PR[90,1] + -25.482;
   1:  PR[91,2] = PR[90,2] + 13.164;
   1:L PR[91] R[100]mm/sec CNT100;
   1:  PR[91,1] = PR[90,1] + -28.038;
   1:  PR[91,2] = PR[90,2] + 8.963;
   1:L PR[91] R[100]mm/sec CNT100;
   1:  PR[91,1] = PR[90,1] + -29.610;
   1:  PR[91,2] = PR[90,2] + 4.399;
   1:L PR[91] R[100]mm/sec CNT100;
   1:  PR[91,1] = PR[90,1] + -29.963;
   1:  PR[91,2] = PR[90,2] + 1.188;
   1:L PR[91] R[100]mm/sec CNT100;
   1:  PR[91,1] = PR[90,1] + -30.116;
   1:  PR[91,2] = PR[90,2] + -0.407;
   1:L PR[91] R[100]mm/sec CNT100;
   1:  PR[91,1] = PR[90,1] + -29.842;
   1:  PR[91,2] = PR[90,2] + -2.902;
   1:L PR[91] R[100]mm/sec CNT100;
   1:  PR[91,1] = PR[90,1] + -29.785;
   1:  PR[91,2] = PR[90,2] + -3.662;
   1:L PR[91] R[100]mm/sec CNT100;
   1:  PR[91,1] = PR[90,1] + -29.611;
   1:  PR[91,2] = PR[90,2] + -5.245;
   1:L PR[91] R[100]mm/sec CNT100;
   1:  PR[91,1] = PR[90,1] + -28.038;
   1:  PR[91,2] = PR[90,2] + -9.810;
   1:L PR[91] R[100]mm/sec CNT100;
   1:  PR[91,1] = PR[90,1] + -25.482;
   1:  PR[91,2] = PR[90,2] + -14.011;
   1:L PR[91] R[100]mm/sec CNT100;
   1:  PR[91,1] = PR[90,1] + -22.051;
   1:  PR[91,2] = PR[90,2] + -17.597;
   1:L PR[91] R[100]mm/sec CNT100;
   1:  PR[91,1] = PR[90,1] + -17.883;
   1:  PR[91,2] = PR[90,2] + -20.408;
   1:L PR[91] R[100]mm/sec CNT100;
   1:  PR[91,1] = PR[90,1] + -15.538;
   1:  PR[91,2] = PR[90,2] + -21.360;
   1:L PR[91] R[100]mm/sec CNT100;
   1:  PR[91,1] = PR[90,1] + -13.176;
   1:  PR[91,2] = PR[90,2] + -22.296;
   1:L PR[91] R[100]mm/sec CNT100;
   1:  PR[91,1] = PR[90,1] + -10.889;
   1:  PR[91,2] = PR[90,2] + -22.702;
   1:L PR[91] R[100]mm/sec CNT100;
   1:  PR[91,1] = PR[90,1] + -8.140;
   1:  PR[91,2] = PR[90,2] + -23.154;
   1:L PR[91] R[100]mm/sec CNT100;
   1:  PR[91,1] = PR[90,1] + -6.032;
   1:  PR[91,2] = PR[90,2] + -23.081;
   1:L PR[91] R[100]mm/sec CNT100;
   1:  PR[91,1] = PR[90,1] + -3.037;
   1:  PR[91,2] = PR[90,2] + -22.931;
   1:L PR[91] R[100]mm/sec CNT100;
   1:  PR[91,1] = PR[90,1] + -0.889;
   1:  PR[91,2] = PR[90,2] + -22.434;
   1:L PR[91] R[100]mm/sec CNT100;
   1:  PR[91,1] = PR[90,1] + 0.425;
   1:  PR[91,2] = PR[90,2] + -22.443;
   1:L PR[91] R[100]mm/sec CNT100;
   1:  PR[91,1] = PR[90,1] + 2.556;
   1:  PR[91,2] = PR[90,2] + -22.931;
   1:L PR[91] R[100]mm/sec CNT100;
   1:  PR[91,1] = PR[90,1] + 5.553;
   1:  PR[91,2] = PR[90,2] + -23.081;
   1:L PR[91] R[100]mm/sec CNT100;
   1:  PR[91,1] = PR[90,1] + 7.661;
   1:  PR[91,2] = PR[90,2] + -23.154;
   1:L PR[91] R[100]mm/sec CNT100;
   1:  PR[91,1] = PR[90,1] + 10.409;
   1:  PR[91,2] = PR[90,2] + -22.702;
   1:L PR[91] R[100]mm/sec CNT100;
   1:  PR[91,1] = PR[90,1] + 12.697;
   1:  PR[91,2] = PR[90,2] + -22.295;
   1:L PR[91] R[100]mm/sec CNT100;
   1:  PR[91,1] = PR[90,1] + 15.060;
   1:  PR[91,2] = PR[90,2] + -21.359;
   1:L PR[91] R[100]mm/sec CNT100;
   1:  PR[91,1] = PR[90,1] + 17.404;
   1:  PR[91,2] = PR[90,2] + -20.408;
   1:L PR[91] R[100]mm/sec CNT100;
   1:  PR[91,1] = PR[90,1] + 21.571;
   1:  PR[91,2] = PR[90,2] + -17.598;
   1:L PR[91] R[100]mm/sec CNT100;
   1:  PR[91,1] = PR[90,1] + 25.003;
   1:  PR[91,2] = PR[90,2] + -14.007;
   1:L PR[91] R[100]mm/sec CNT100;
   1:  PR[91,1] = PR[90,1] + 27.559;
   1:  PR[91,2] = PR[90,2] + -9.809;
   1:L PR[91] R[100]mm/sec CNT100;
   1:  PR[91,1] = PR[90,1] + 29.131;
   1:  PR[91,2] = PR[90,2] + -5.253;
   1:L PR[91] R[100]mm/sec CNT100;
   1:  PR[91,1] = PR[90,1] + 29.484;
   1:  PR[91,2] = PR[90,2] + -2.036;
   1:L PR[91] R[100]mm/sec CNT100;
   1:  PR[91,1] = PR[90,1] + 29.637;
   1:  PR[91,2] = PR[90,2] + -0.440;
   1:L PR[91] R[100]mm/sec CNT100;
   1:  PR[91,1] = PR[90,1] + 29.362;
   1:  PR[91,2] = PR[90,2] + 2.061;
   1:L PR[91] R[100]mm/sec CNT100;
   1:  PR[91,1] = PR[90,1] + 29.305;
   1:  PR[91,2] = PR[90,2] + 2.822;
   1:L PR[91] R[100]mm/sec CNT100;
   1:  PR[91,1] = PR[90,1] + 29.131;
   1:  PR[91,2] = PR[90,2] + 4.406;
   1:L PR[91] R[100]mm/sec CNT100;
   1:  PR[91,1] = PR[90,1] + 27.559;
   1:  PR[91,2] = PR[90,2] + 8.962;
   1:L PR[91] R[100]mm/sec CNT100;
   1:  PR[91,1] = PR[90,1] + 25.002;
   1:  PR[91,2] = PR[90,2] + 13.161;
   1:L PR[91] R[100]mm/sec CNT100;
   1:  PR[91,1] = PR[90,1] + 21.570;
   1:  PR[91,2] = PR[90,2] + 16.751;
   1:L PR[91] R[100]mm/sec CNT100;
   1:  PR[91,1] = PR[90,1] + 17.403;
   1:  PR[91,2] = PR[90,2] + 19.561;
   1:L PR[91] R[100]mm/sec CNT100;
   1:  PR[91,1] = PR[90,1] + 15.059;
   1:  PR[91,2] = PR[90,2] + 20.512;
   1:L PR[91] R[100]mm/sec CNT100;
   1:  PR[91,1] = PR[90,1] + 12.695;
   1:  PR[91,2] = PR[90,2] + 21.448;
   1:L PR[91] R[100]mm/sec CNT100;
   1:  PR[91,1] = PR[90,1] + 10.407;
   1:  PR[91,2] = PR[90,2] + 21.855;
   1:L PR[91] R[100]mm/sec CNT100;
   1:  PR[91,1] = PR[90,1] + 7.659;
   1:  PR[91,2] = PR[90,2] + 22.307;
   1:L PR[91] R[100]mm/sec CNT100;
   1:  PR[91,1] = PR[90,1] + 5.551;
   1:  PR[91,2] = PR[90,2] + 22.234;
   1:L PR[91] R[100]mm/sec CNT100;
   1:  PR[91,1] = PR[90,1] + 2.557;
   1:  PR[91,2] = PR[90,2] + 22.084;
   1:L PR[91] R[100]mm/sec CNT100;
   1:  PR[91,1] = PR[90,1] + 0.422;
   1:  PR[91,2] = PR[90,2] + 21.596;
   1:L PR[91] R[100]mm/sec CNT100;
   1:  PR[91] = PR[90];
   1:  PR[91,1] = PR[90,1] + -0.861;
   1:  PR[91,2] = PR[90,2] + 21.943;
   1:  PR[91,3] = PR[90,3] + 58.695;
   1:L PR[91] R[100]mm/sec CNT100;
   1:  PR[91,1] = PR[90,1] + -2.490;
   1:  PR[91,2] = PR[90,2] + 22.319;
   1:L PR[91] R[100]mm/sec CNT100;
   1:  PR[91,1] = PR[90,1] + -6.071;
   1:  PR[91,2] = PR[90,2] + 22.498;
   1:L PR[91] R[100]mm/sec CNT100;
   1:  PR[91,1] = PR[90,1] + -7.625;
   1:  PR[91,2] = PR[90,2] + 22.552;
   1:L PR[91] R[100]mm/sec CNT100;
   1:  PR[91,1] = PR[90,1] + -10.979;
   1:  PR[91,2] = PR[90,2] + 22.001;
   1:L PR[91] R[100]mm/sec CNT100;
   1:  PR[91,1] = PR[90,1] + -12.707;
   1:  PR[91,2] = PR[90,2] + 21.694;
   1:L PR[91] R[100]mm/sec CNT100;
   1:  PR[91,1] = PR[90,1] + -15.654;
   1:  PR[91,2] = PR[90,2] + 20.527;
   1:L PR[91] R[100]mm/sec CNT100;
   1:  PR[91,1] = PR[90,1] + -17.461;
   1:  PR[91,2] = PR[90,2] + 19.793;
   1:L PR[91] R[100]mm/sec CNT100;
   1:  PR[91,1] = PR[90,1] + -21.673;
   1:  PR[91,2] = PR[90,2] + 16.955;
   1:L PR[91] R[100]mm/sec CNT100;
   1:  PR[91,1] = PR[90,1] + -25.141;
   1:  PR[91,2] = PR[90,2] + 13.331;
   1:L PR[91] R[100]mm/sec CNT100;
   1:  PR[91,1] = PR[90,1] + -27.727;
   1:  PR[91,2] = PR[90,2] + 9.082;
   1:L PR[91] R[100]mm/sec CNT100;
   1:  PR[91,1] = PR[90,1] + -29.318;
   1:  PR[91,2] = PR[90,2] + 4.458;
   1:L PR[91] R[100]mm/sec CNT100;
   1:  PR[91,1] = PR[90,1] + -29.600;
   1:  PR[91,2] = PR[90,2] + 1.887;
   1:L PR[91] R[100]mm/sec CNT100;
   1:  PR[91,1] = PR[90,1] + -29.821;
   1:  PR[91,2] = PR[90,2] + -0.407;
   1:L PR[91] R[100]mm/sec CNT100;
   1:  PR[91,1] = PR[90,1] + -29.645;
   1:  PR[91,2] = PR[90,2] + -1.999;
   1:L PR[91] R[100]mm/sec CNT100;
   1:  PR[91,1] = PR[90,1] + -29.568;
   1:  PR[91,2] = PR[90,2] + -3.034;
   1:L PR[91] R[100]mm/sec CNT100;
   1:  PR[91,1] = PR[90,1] + -29.318;
   1:  PR[91,2] = PR[90,2] + -5.304;
   1:L PR[91] R[100]mm/sec CNT100;
   1:  PR[91,1] = PR[90,1] + -27.727;
   1:  PR[91,2] = PR[90,2] + -9.929;
   1:L PR[91] R[100]mm/sec CNT100;
   1:  PR[91,1] = PR[90,1] + -25.142;
   1:  PR[91,2] = PR[90,2] + -14.178;
   1:L PR[91] R[100]mm/sec CNT100;
   1:  PR[91,1] = PR[90,1] + -21.673;
   1:  PR[91,2] = PR[90,2] + -17.802;
   1:L PR[91] R[100]mm/sec CNT100;
   1:  PR[91,1] = PR[90,1] + -17.462;
   1:  PR[91,2] = PR[90,2] + -20.640;
   1:L PR[91] R[100]mm/sec CNT100;
   1:  PR[91,1] = PR[90,1] + -15.655;
   1:  PR[91,2] = PR[90,2] + -21.373;
   1:L PR[91] R[100]mm/sec CNT100;
   1:  PR[91,1] = PR[90,1] + -12.709;
   1:  PR[91,2] = PR[90,2] + -22.540;
   1:L PR[91] R[100]mm/sec CNT100;
   1:  PR[91,1] = PR[90,1] + -10.981;
   1:  PR[91,2] = PR[90,2] + -22.847;
   1:L PR[91] R[100]mm/sec CNT100;
   1:  PR[91,1] = PR[90,1] + -7.627;
   1:  PR[91,2] = PR[90,2] + -23.399;
   1:L PR[91] R[100]mm/sec CNT100;
   1:  PR[91,1] = PR[90,1] + -6.073;
   1:  PR[91,2] = PR[90,2] + -23.345;
   1:L PR[91] R[100]mm/sec CNT100;
   1:  PR[91,1] = PR[90,1] + -2.489;
   1:  PR[91,2] = PR[90,2] + -23.166;
   1:L PR[91] R[100]mm/sec CNT100;
   1:  PR[91,1] = PR[90,1] + -0.860;
   1:  PR[91,2] = PR[90,2] + -22.789;
   1:L PR[91] R[100]mm/sec CNT100;
   1:  PR[91,1] = PR[90,1] + 0.392;
   1:  PR[91,2] = PR[90,2] + -22.796;
   1:L PR[91] R[100]mm/sec CNT100;
   1:  PR[91,1] = PR[90,1] + 2.007;
   1:  PR[91,2] = PR[90,2] + -23.166;
   1:L PR[91] R[100]mm/sec CNT100;
   1:  PR[91,1] = PR[90,1] + 5.594;
   1:  PR[91,2] = PR[90,2] + -23.345;
   1:L PR[91] R[100]mm/sec CNT100;
   1:  PR[91,1] = PR[90,1] + 7.148;
   1:  PR[91,2] = PR[90,2] + -23.399;
   1:L PR[91] R[100]mm/sec CNT100;
   1:  PR[91,1] = PR[90,1] + 10.501;
   1:  PR[91,2] = PR[90,2] + -22.847;
   1:L PR[91] R[100]mm/sec CNT100;
   1:  PR[91,1] = PR[90,1] + 12.229;
   1:  PR[91,2] = PR[90,2] + -22.540;
   1:L PR[91] R[100]mm/sec CNT100;
   1:  PR[91,1] = PR[90,1] + 15.176;
   1:  PR[91,2] = PR[90,2] + -21.373;
   1:L PR[91] R[100]mm/sec CNT100;
   1:  PR[91,1] = PR[90,1] + 16.983;
   1:  PR[91,2] = PR[90,2] + -20.640;
   1:L PR[91] R[100]mm/sec CNT100;
   1:  PR[91,1] = PR[90,1] + 21.193;
   1:  PR[91,2] = PR[90,2] + -17.803;
   1:L PR[91] R[100]mm/sec CNT100;
   1:  PR[91,1] = PR[90,1] + 24.662;
   1:  PR[91,2] = PR[90,2] + -14.174;
   1:L PR[91] R[100]mm/sec CNT100;
   1:  PR[91,1] = PR[90,1] + 27.248;
   1:  PR[91,2] = PR[90,2] + -9.928;
   1:L PR[91] R[100]mm/sec CNT100;
   1:  PR[91,1] = PR[90,1] + 28.838;
   1:  PR[91,2] = PR[90,2] + -5.311;
   1:L PR[91] R[100]mm/sec CNT100;
   1:  PR[91,1] = PR[90,1] + 29.121;
   1:  PR[91,2] = PR[90,2] + -2.735;
   1:L PR[91] R[100]mm/sec CNT100;
   1:  PR[91,1] = PR[90,1] + 29.341;
   1:  PR[91,2] = PR[90,2] + -0.440;
   1:L PR[91] R[100]mm/sec CNT100;
   1:  PR[91,1] = PR[90,1] + 29.165;
   1:  PR[91,2] = PR[90,2] + 1.156;
   1:L PR[91] R[100]mm/sec CNT100;
   1:  PR[91,1] = PR[90,1] + 29.088;
   1:  PR[91,2] = PR[90,2] + 2.193;
   1:L PR[91] R[100]mm/sec CNT100;
   1:  PR[91,1] = PR[90,1] + 28.838;
   1:  PR[91,2] = PR[90,2] + 4.464;
   1:L PR[91] R[100]mm/sec CNT100;
   1:  PR[91,1] = PR[90,1] + 27.247;
   1:  PR[91,2] = PR[90,2] + 9.081;
   1:L PR[91] R[100]mm/sec CNT100;
   1:  PR[91,1] = PR[90,1] + 24.662;
   1:  PR[91,2] = PR[90,2] + 13.328;
   1:L PR[91] R[100]mm/sec CNT100;
   1:  PR[91,1] = PR[90,1] + 21.193;
   1:  PR[91,2] = PR[90,2] + 16.956;
   1:L PR[91] R[100]mm/sec CNT100;
   1:  PR[91,1] = PR[90,1] + 16.982;
   1:  PR[91,2] = PR[90,2] + 19.793;
   1:L PR[91] R[100]mm/sec CNT100;
   1:  PR[91,1] = PR[90,1] + 15.175;
   1:  PR[91,2] = PR[90,2] + 20.526;
   1:L PR[91] R[100]mm/sec CNT100;
   1:  PR[91,1] = PR[90,1] + 12.228;
   1:  PR[91,2] = PR[90,2] + 21.693;
   1:L PR[91] R[100]mm/sec CNT100;
   1:  PR[91,1] = PR[90,1] + 10.499;
   1:  PR[91,2] = PR[90,2] + 22.000;
   1:L PR[91] R[100]mm/sec CNT100;
   1:  PR[91,1] = PR[90,1] + 7.146;
   1:  PR[91,2] = PR[90,2] + 22.552;
   1:L PR[91] R[100]mm/sec CNT100;
   1:  PR[91,1] = PR[90,1] + 5.592;
   1:  PR[91,2] = PR[90,2] + 22.498;
   1:L PR[91] R[100]mm/sec CNT100;
   1:  PR[91,1] = PR[90,1] + 2.009;
   1:  PR[91,2] = PR[90,2] + 22.319;
   1:L PR[91] R[100]mm/sec CNT100;
   1:  PR[91,1] = PR[90,1] + 0.390;
   1:  PR[91,2] = PR[90,2] + 21.948;
   1:L PR[91] R[100]mm/sec CNT100;
   1:  PR[91] = PR[90];
   1:  PR[91,1] = PR[90,1] + -0.831;
   1:  PR[91,2] = PR[90,2] + 22.298;
   1:  PR[91,3] = PR[90,3] + 59.995;
   1:L PR[91] R[100]mm/sec CNT100;
   1:  PR[91,1] = PR[90,1] + -1.942;
   1:  PR[91,2] = PR[90,2] + 22.554;
   1:L PR[91] R[100]mm/sec CNT100;
   1:  PR[91,1] = PR[90,1] + -6.112;
   1:  PR[91,2] = PR[90,2] + 22.762;
   1:L PR[91] R[100]mm/sec CNT100;
   1:  PR[91,1] = PR[90,1] + -7.111;
   1:  PR[91,2] = PR[90,2] + 22.796;
   1:L PR[91] R[100]mm/sec CNT100;
   1:  PR[91,1] = PR[90,1] + -11.070;
   1:  PR[91,2] = PR[90,2] + 22.146;
   1:L PR[91] R[100]mm/sec CNT100;
   1:  PR[91,1] = PR[90,1] + -12.236;
   1:  PR[91,2] = PR[90,2] + 21.939;
   1:L PR[91] R[100]mm/sec CNT100;
   1:  PR[91,1] = PR[90,1] + -17.046;
   1:  PR[91,2] = PR[90,2] + 20.021;
   1:L PR[91] R[100]mm/sec CNT100;
   1:  PR[91,1] = PR[90,1] + -21.295;
   1:  PR[91,2] = PR[90,2] + 17.160;
   1:L PR[91] R[100]mm/sec CNT100;
   1:  PR[91,1] = PR[90,1] + -24.801;
   1:  PR[91,2] = PR[90,2] + 13.498;
   1:L PR[91] R[100]mm/sec CNT100;
   1:  PR[91,1] = PR[90,1] + -27.415;
   1:  PR[91,2] = PR[90,2] + 9.202;
   1:L PR[91] R[100]mm/sec CNT100;
   1:  PR[91,1] = PR[90,1] + -29.025;
   1:  PR[91,2] = PR[90,2] + 4.517;
   1:L PR[91] R[100]mm/sec CNT100;
   1:  PR[91,1] = PR[90,1] + -29.238;
   1:  PR[91,2] = PR[90,2] + 2.585;
   1:L PR[91] R[100]mm/sec CNT100;
   1:  PR[91,1] = PR[90,1] + -29.525;
   1:  PR[91,2] = PR[90,2] + -0.407;
   1:L PR[91] R[100]mm/sec CNT100;
   1:  PR[91,1] = PR[90,1] + -29.449;
   1:  PR[91,2] = PR[90,2] + -1.097;
   1:L PR[91] R[100]mm/sec CNT100;
   1:  PR[91,1] = PR[90,1] + -29.351;
   1:  PR[91,2] = PR[90,2] + -2.407;
   1:L PR[91] R[100]mm/sec CNT100;
   1:  PR[91,1] = PR[90,1] + -29.025;
   1:  PR[91,2] = PR[90,2] + -5.363;
   1:L PR[91] R[100]mm/sec CNT100;
   1:  PR[91,1] = PR[90,1] + -27.415;
   1:  PR[91,2] = PR[90,2] + -10.049;
   1:L PR[91] R[100]mm/sec CNT100;
   1:  PR[91,1] = PR[90,1] + -24.801;
   1:  PR[91,2] = PR[90,2] + -14.344;
   1:L PR[91] R[100]mm/sec CNT100;
   1:  PR[91,1] = PR[90,1] + -21.296;
   1:  PR[91,2] = PR[90,2] + -18.007;
   1:L PR[91] R[100]mm/sec CNT100;
   1:  PR[91,1] = PR[90,1] + -17.047;
   1:  PR[91,2] = PR[90,2] + -20.867;
   1:L PR[91] R[100]mm/sec CNT100;
   1:  PR[91,1] = PR[90,1] + -12.239;
   1:  PR[91,2] = PR[90,2] + -22.785;
   1:L PR[91] R[100]mm/sec CNT100;
   1:  PR[91,1] = PR[90,1] + -11.073;
   1:  PR[91,2] = PR[90,2] + -22.992;
   1:L PR[91] R[100]mm/sec CNT100;
   1:  PR[91,1] = PR[90,1] + -7.114;
   1:  PR[91,2] = PR[90,2] + -23.644;
   1:L PR[91] R[100]mm/sec CNT100;
   1:  PR[91,1] = PR[90,1] + -6.114;
   1:  PR[91,2] = PR[90,2] + -23.609;
   1:L PR[91] R[100]mm/sec CNT100;
   1:  PR[91,1] = PR[90,1] + -1.940;
   1:  PR[91,2] = PR[90,2] + -23.400;
   1:L PR[91] R[100]mm/sec CNT100;
   1:  PR[91,1] = PR[90,1] + -0.831;
   1:  PR[91,2] = PR[90,2] + -23.144;
   1:L PR[91] R[100]mm/sec CNT100;
   1:  PR[91,1] = PR[90,1] + 0.359;
   1:  PR[91,2] = PR[90,2] + -23.149;
   1:L PR[91] R[100]mm/sec CNT100;
   1:  PR[91,1] = PR[90,1] + 1.458;
   1:  PR[91,2] = PR[90,2] + -23.400;
   1:L PR[91] R[100]mm/sec CNT100;
   1:  PR[91,1] = PR[90,1] + 5.635;
   1:  PR[91,2] = PR[90,2] + -23.609;
   1:L PR[91] R[100]mm/sec CNT100;
   1:  PR[91,1] = PR[90,1] + 6.635;
   1:  PR[91,2] = PR[90,2] + -23.644;
   1:L PR[91] R[100]mm/sec CNT100;
   1:  PR[91,1] = PR[90,1] + 10.593;
   1:  PR[91,2] = PR[90,2] + -22.992;
   1:L PR[91] R[100]mm/sec CNT100;
   1:  PR[91,1] = PR[90,1] + 11.762;
   1:  PR[91,2] = PR[90,2] + -22.784;
   1:L PR[91] R[100]mm/sec CNT100;
   1:  PR[91,1] = PR[90,1] + 15.293;
   1:  PR[91,2] = PR[90,2] + -21.386;
   1:L PR[91] R[100]mm/sec CNT100;
   1:  PR[91,1] = PR[90,1] + 16.562;
   1:  PR[91,2] = PR[90,2] + -20.871;
   1:L PR[91] R[100]mm/sec CNT100;
   1:  PR[91,1] = PR[90,1] + 20.816;
   1:  PR[91,2] = PR[90,2] + -18.008;
   1:L PR[91] R[100]mm/sec CNT100;
   1:  PR[91,1] = PR[90,1] + 24.322;
   1:  PR[91,2] = PR[90,2] + -14.342;
   1:L PR[91] R[100]mm/sec CNT100;
   1:  PR[91,1] = PR[90,1] + 26.936;
   1:  PR[91,2] = PR[90,2] + -10.048;
   1:L PR[91] R[100]mm/sec CNT100;
   1:  PR[91,1] = PR[90,1] + 28.546;
   1:  PR[91,2] = PR[90,2] + -5.370;
   1:L PR[91] R[100]mm/sec CNT100;
   1:  PR[91,1] = PR[90,1] + 28.758;
   1:  PR[91,2] = PR[90,2] + -3.433;
   1:L PR[91] R[100]mm/sec CNT100;
   1:  PR[91,1] = PR[90,1] + 29.045;
   1:  PR[91,2] = PR[90,2] + -0.440;
   1:L PR[91] R[100]mm/sec CNT100;
   1:  PR[91,1] = PR[90,1] + 28.969;
   1:  PR[91,2] = PR[90,2] + 0.252;
   1:L PR[91] R[100]mm/sec CNT100;
   1:  PR[91,1] = PR[90,1] + 28.872;
   1:  PR[91,2] = PR[90,2] + 1.564;
   1:L PR[91] R[100]mm/sec CNT100;
   1:  PR[91,1] = PR[90,1] + 28.546;
   1:  PR[91,2] = PR[90,2] + 4.522;
   1:L PR[91] R[100]mm/sec CNT100;
   1:  PR[91,1] = PR[90,1] + 26.936;
   1:  PR[91,2] = PR[90,2] + 9.201;
   1:L PR[91] R[100]mm/sec CNT100;
   1:  PR[91,1] = PR[90,1] + 24.321;
   1:  PR[91,2] = PR[90,2] + 13.495;
   1:L PR[91] R[100]mm/sec CNT100;
   1:  PR[91,1] = PR[90,1] + 20.815;
   1:  PR[91,2] = PR[90,2] + 17.161;
   1:L PR[91] R[100]mm/sec CNT100;
   1:  PR[91,1] = PR[90,1] + 16.567;
   1:  PR[91,2] = PR[90,2] + 20.021;
   1:L PR[91] R[100]mm/sec CNT100;
   1:  PR[91,1] = PR[90,1] + 11.757;
   1:  PR[91,2] = PR[90,2] + 21.938;
   1:L PR[91] R[100]mm/sec CNT100;
   1:  PR[91,1] = PR[90,1] + 10.590;
   1:  PR[91,2] = PR[90,2] + 22.146;
   1:L PR[91] R[100]mm/sec CNT100;
   1:  PR[91,1] = PR[90,1] + 6.632;
   1:  PR[91,2] = PR[90,2] + 22.797;
   1:L PR[91] R[100]mm/sec CNT100;
   1:  PR[91,1] = PR[90,1] + 5.632;
   1:  PR[91,2] = PR[90,2] + 22.762;
   1:L PR[91] R[100]mm/sec CNT100;
   1:  PR[91,1] = PR[90,1] + 1.461;
   1:  PR[91,2] = PR[90,2] + 22.554;
   1:L PR[91] R[100]mm/sec CNT100;
   1:  PR[91,1] = PR[90,1] + 0.358;
   1:  PR[91,2] = PR[90,2] + 22.301;
   1:L PR[91] R[100]mm/sec CNT100;
   1:  PR[91] = PR[90];
   1:  PR[91,1] = PR[90,1] + -0.802;
   1:  PR[91,2] = PR[90,2] + 22.652;
   1:  PR[91,3] = PR[90,3] + 61.295;
   1:L PR[91] R[100]mm/sec CNT100;
   1:  PR[91,1] = PR[90,1] + -1.391;
   1:  PR[91,2] = PR[90,2] + 22.788;
   1:L PR[91] R[100]mm/sec CNT100;
   1:  PR[91,1] = PR[90,1] + -6.612;
   1:  PR[91,2] = PR[90,2] + 23.038;
   1:L PR[91] R[100]mm/sec CNT100;
   1:  PR[91,1] = PR[90,1] + -11.782;
   1:  PR[91,2] = PR[90,2] + 22.178;
   1:L PR[91] R[100]mm/sec CNT100;
   1:  PR[91,1] = PR[90,1] + -16.625;
   1:  PR[91,2] = PR[90,2] + 20.252;
   1:L PR[91] R[100]mm/sec CNT100;
   1:  PR[91,1] = PR[90,1] + -20.917;
   1:  PR[91,2] = PR[90,2] + 17.365;
   1:L PR[91] R[100]mm/sec CNT100;
   1:  PR[91,1] = PR[90,1] + -24.460;
   1:  PR[91,2] = PR[90,2] + 13.665;
   1:L PR[91] R[100]mm/sec CNT100;
   1:  PR[91,1] = PR[90,1] + -27.104;
   1:  PR[91,2] = PR[90,2] + 9.321;
   1:L PR[91] R[100]mm/sec CNT100;
   1:  PR[91,1] = PR[90,1] + -28.733;
   1:  PR[91,2] = PR[90,2] + 4.576;
   1:L PR[91] R[100]mm/sec CNT100;
   1:  PR[91,1] = PR[90,1] + -28.875;
   1:  PR[91,2] = PR[90,2] + 3.284;
   1:L PR[91] R[100]mm/sec CNT100;
   1:  PR[91,1] = PR[90,1] + -29.233;
   1:  PR[91,2] = PR[90,2] + -0.450;
   1:L PR[91] R[100]mm/sec CNT100;
   1:  PR[91,1] = PR[90,1] + -29.134;
   1:  PR[91,2] = PR[90,2] + -1.779;
   1:L PR[91] R[100]mm/sec CNT100;
   1:  PR[91,1] = PR[90,1] + -28.733;
   1:  PR[91,2] = PR[90,2] + -5.422;
   1:L PR[91] R[100]mm/sec CNT100;
   1:  PR[91,1] = PR[90,1] + -27.104;
   1:  PR[91,2] = PR[90,2] + -10.168;
   1:L PR[91] R[100]mm/sec CNT100;
   1:  PR[91,1] = PR[90,1] + -24.461;
   1:  PR[91,2] = PR[90,2] + -14.511;
   1:L PR[91] R[100]mm/sec CNT100;
   1:  PR[91,1] = PR[90,1] + -20.918;
   1:  PR[91,2] = PR[90,2] + -18.211;
   1:L PR[91] R[100]mm/sec CNT100;
   1:  PR[91,1] = PR[90,1] + -16.627;
   1:  PR[91,2] = PR[90,2] + -21.098;
   1:L PR[91] R[100]mm/sec CNT100;
   1:  PR[91,1] = PR[90,1] + -11.784;
   1:  PR[91,2] = PR[90,2] + -23.025;
   1:L PR[91] R[100]mm/sec CNT100;
   1:  PR[91,1] = PR[90,1] + -6.615;
   1:  PR[91,2] = PR[90,2] + -23.886;
   1:L PR[91] R[100]mm/sec CNT100;
   1:  PR[91,1] = PR[90,1] + -1.389;
   1:  PR[91,2] = PR[90,2] + -23.634;
   1:L PR[91] R[100]mm/sec CNT100;
   1:  PR[91,1] = PR[90,1] + -0.802;
   1:  PR[91,2] = PR[90,2] + -23.499;
   1:L PR[91] R[100]mm/sec CNT100;
   1:  PR[91,1] = PR[90,1] + 0.325;
   1:  PR[91,2] = PR[90,2] + -23.501;
   1:L PR[91] R[100]mm/sec CNT100;
   1:  PR[91,1] = PR[90,1] + 0.907;
   1:  PR[91,2] = PR[90,2] + -23.634;
   1:L PR[91] R[100]mm/sec CNT100;
   1:  PR[91,1] = PR[90,1] + 6.136;
   1:  PR[91,2] = PR[90,2] + -23.886;
   1:L PR[91] R[100]mm/sec CNT100;
   1:  PR[91,1] = PR[90,1] + 11.307;
   1:  PR[91,2] = PR[90,2] + -23.024;
   1:L PR[91] R[100]mm/sec CNT100;
   1:  PR[91,1] = PR[90,1] + 15.410;
   1:  PR[91,2] = PR[90,2] + -21.399;
   1:L PR[91] R[100]mm/sec CNT100;
   1:  PR[91,1] = PR[90,1] + 16.142;
   1:  PR[91,2] = PR[90,2] + -21.102;
   1:L PR[91] R[100]mm/sec CNT100;
   1:  PR[91,1] = PR[90,1] + 20.438;
   1:  PR[91,2] = PR[90,2] + -18.212;
   1:L PR[91] R[100]mm/sec CNT100;
   1:  PR[91,1] = PR[90,1] + 23.981;
   1:  PR[91,2] = PR[90,2] + -14.509;
   1:L PR[91] R[100]mm/sec CNT100;
   1:  PR[91,1] = PR[90,1] + 26.625;
   1:  PR[91,2] = PR[90,2] + -10.167;
   1:L PR[91] R[100]mm/sec CNT100;
   1:  PR[91,1] = PR[90,1] + 28.253;
   1:  PR[91,2] = PR[90,2] + -5.428;
   1:L PR[91] R[100]mm/sec CNT100;
   1:  PR[91,1] = PR[90,1] + 28.395;
   1:  PR[91,2] = PR[90,2] + -4.133;
   1:L PR[91] R[100]mm/sec CNT100;
   1:  PR[91,1] = PR[90,1] + 28.754;
   1:  PR[91,2] = PR[90,2] + -0.398;
   1:L PR[91] R[100]mm/sec CNT100;
   1:  PR[91,1] = PR[90,1] + 28.655;
   1:  PR[91,2] = PR[90,2] + 0.936;
   1:L PR[91] R[100]mm/sec CNT100;
   1:  PR[91,1] = PR[90,1] + 28.253;
   1:  PR[91,2] = PR[90,2] + 4.580;
   1:L PR[91] R[100]mm/sec CNT100;
   1:  PR[91,1] = PR[90,1] + 26.624;
   1:  PR[91,2] = PR[90,2] + 9.321;
   1:L PR[91] R[100]mm/sec CNT100;
   1:  PR[91,1] = PR[90,1] + 23.981;
   1:  PR[91,2] = PR[90,2] + 13.662;
   1:L PR[91] R[100]mm/sec CNT100;
   1:  PR[91,1] = PR[90,1] + 20.437;
   1:  PR[91,2] = PR[90,2] + 17.366;
   1:L PR[91] R[100]mm/sec CNT100;
   1:  PR[91,1] = PR[90,1] + 16.140;
   1:  PR[91,2] = PR[90,2] + 20.256;
   1:L PR[91] R[100]mm/sec CNT100;
   1:  PR[91,1] = PR[90,1] + 15.408;
   1:  PR[91,2] = PR[90,2] + 20.553;
   1:L PR[91] R[100]mm/sec CNT100;
   1:  PR[91,1] = PR[90,1] + 11.305;
   1:  PR[91,2] = PR[90,2] + 22.178;
   1:L PR[91] R[100]mm/sec CNT100;
   1:  PR[91,1] = PR[90,1] + 6.132;
   1:  PR[91,2] = PR[90,2] + 23.039;
   1:L PR[91] R[100]mm/sec CNT100;
   1:  PR[91,1] = PR[90,1] + 0.910;
   1:  PR[91,2] = PR[90,2] + 22.788;
   1:L PR[91] R[100]mm/sec CNT100;
   1:  PR[91,1] = PR[90,1] + 0.325;
   1:  PR[91,2] = PR[90,2] + 22.654;
   1:L PR[91] R[100]mm/sec CNT100;
   1:  PR[91] = PR[90];
   1:  PR[91,1] = PR[90,1] + -0.555;
   1:  PR[91,2] = PR[90,2] + 23.006;
   1:  PR[91,3] = PR[90,3] + 62.595;
   1:L PR[91] R[100]mm/sec CNT100;
   1:  PR[91,1] = PR[90,1] + -6.102;
   1:  PR[91,2] = PR[90,2] + 23.283;
   1:L PR[91] R[100]mm/sec CNT100;
   1:  PR[91,1] = PR[90,1] + -11.317;
   1:  PR[91,2] = PR[90,2] + 22.422;
   1:L PR[91] R[100]mm/sec CNT100;
   1:  PR[91,1] = PR[90,1] + -16.205;
   1:  PR[91,2] = PR[90,2] + 20.483;
   1:L PR[91] R[100]mm/sec CNT100;
   1:  PR[91,1] = PR[90,1] + -20.539;
   1:  PR[91,2] = PR[90,2] + 17.570;
   1:L PR[91] R[100]mm/sec CNT100;
   1:  PR[91,1] = PR[90,1] + -24.120;
   1:  PR[91,2] = PR[90,2] + 13.832;
   1:L PR[91] R[100]mm/sec CNT100;
   1:  PR[91,1] = PR[90,1] + -26.792;
   1:  PR[91,2] = PR[90,2] + 9.441;
   1:L PR[91] R[100]mm/sec CNT100;
   1:  PR[91,1] = PR[90,1] + -28.436;
   1:  PR[91,2] = PR[90,2] + 4.646;
   1:L PR[91] R[100]mm/sec CNT100;
   1:  PR[91,1] = PR[90,1] + -28.736;
   1:  PR[91,2] = PR[90,2] + 1.645;
   1:L PR[91] R[100]mm/sec CNT100;
   1:  PR[91,1] = PR[90,1] + -28.968;
   1:  PR[91,2] = PR[90,2] + -0.466;
   1:L PR[91] R[100]mm/sec CNT100;
   1:  PR[91,1] = PR[90,1] + -28.917;
   1:  PR[91,2] = PR[90,2] + -1.152;
   1:L PR[91] R[100]mm/sec CNT100;
   1:  PR[91,1] = PR[90,1] + -28.440;
   1:  PR[91,2] = PR[90,2] + -5.481;
   1:L PR[91] R[100]mm/sec CNT100;
   1:  PR[91,1] = PR[90,1] + -26.793;
   1:  PR[91,2] = PR[90,2] + -10.287;
   1:L PR[91] R[100]mm/sec CNT100;
   1:  PR[91,1] = PR[90,1] + -24.120;
   1:  PR[91,2] = PR[90,2] + -14.678;
   1:L PR[91] R[100]mm/sec CNT100;
   1:  PR[91,1] = PR[90,1] + -20.540;
   1:  PR[91,2] = PR[90,2] + -18.416;
   1:L PR[91] R[100]mm/sec CNT100;
   1:  PR[91,1] = PR[90,1] + -16.207;
   1:  PR[91,2] = PR[90,2] + -21.329;
   1:L PR[91] R[100]mm/sec CNT100;
   1:  PR[91,1] = PR[90,1] + -11.320;
   1:  PR[91,2] = PR[90,2] + -23.269;
   1:L PR[91] R[100]mm/sec CNT100;
   1:  PR[91,1] = PR[90,1] + -6.105;
   1:  PR[91,2] = PR[90,2] + -24.130;
   1:L PR[91] R[100]mm/sec CNT100;
   1:  PR[91,1] = PR[90,1] + -0.559;
   1:  PR[91,2] = PR[90,2] + -23.853;
   1:L PR[91] R[100]mm/sec CNT100;
   1:  PR[91,1] = PR[90,1] + 0.080;
   1:L PR[91] R[100]mm/sec CNT100;
   1:  PR[91,1] = PR[90,1] + 5.626;
   1:  PR[91,2] = PR[90,2] + -24.130;
   1:L PR[91] R[100]mm/sec CNT100;
   1:  PR[91,1] = PR[90,1] + 10.841;
   1:  PR[91,2] = PR[90,2] + -23.268;
   1:L PR[91] R[100]mm/sec CNT100;
   1:  PR[91,1] = PR[90,1] + 15.728;
   1:  PR[91,2] = PR[90,2] + -21.329;
   1:L PR[91] R[100]mm/sec CNT100;
   1:  PR[91,1] = PR[90,1] + 20.060;
   1:  PR[91,2] = PR[90,2] + -18.417;
   1:L PR[91] R[100]mm/sec CNT100;
   1:  PR[91,1] = PR[90,1] + 23.641;
   1:  PR[91,2] = PR[90,2] + -14.676;
   1:L PR[91] R[100]mm/sec CNT100;
   1:  PR[91,1] = PR[90,1] + 26.313;
   1:  PR[91,2] = PR[90,2] + -10.287;
   1:L PR[91] R[100]mm/sec CNT100;
   1:  PR[91,1] = PR[90,1] + 27.957;
   1:  PR[91,2] = PR[90,2] + -5.497;
   1:L PR[91] R[100]mm/sec CNT100;
   1:  PR[91,1] = PR[90,1] + 28.256;
   1:  PR[91,2] = PR[90,2] + -2.494;
   1:L PR[91] R[100]mm/sec CNT100;
   1:  PR[91,1] = PR[90,1] + 28.489;
   1:  PR[91,2] = PR[90,2] + -0.381;
   1:L PR[91] R[100]mm/sec CNT100;
   1:  PR[91,1] = PR[90,1] + 28.438;
   1:  PR[91,2] = PR[90,2] + 0.307;
   1:L PR[91] R[100]mm/sec CNT100;
   1:  PR[91,1] = PR[90,1] + 27.960;
   1:  PR[91,2] = PR[90,2] + 4.639;
   1:L PR[91] R[100]mm/sec CNT100;
   1:  PR[91,1] = PR[90,1] + 26.313;
   1:  PR[91,2] = PR[90,2] + 9.440;
   1:L PR[91] R[100]mm/sec CNT100;
   1:  PR[91,1] = PR[90,1] + 23.640;
   1:  PR[91,2] = PR[90,2] + 13.830;
   1:L PR[91] R[100]mm/sec CNT100;
   1:  PR[91,1] = PR[90,1] + 20.059;
   1:  PR[91,2] = PR[90,2] + 17.571;
   1:L PR[91] R[100]mm/sec CNT100;
   1:  PR[91,1] = PR[90,1] + 15.726;
   1:  PR[91,2] = PR[90,2] + 20.482;
   1:L PR[91] R[100]mm/sec CNT100;
   1:  PR[91,1] = PR[90,1] + 10.838;
   1:  PR[91,2] = PR[90,2] + 22.422;
   1:L PR[91] R[100]mm/sec CNT100;
   1:  PR[91,1] = PR[90,1] + 5.623;
   1:  PR[91,2] = PR[90,2] + 23.283;
   1:L PR[91] R[100]mm/sec CNT100;
   1:  PR[91,1] = PR[90,1] + 0.080;
   1:  PR[91,2] = PR[90,2] + 23.006;
   1:L PR[91] R[100]mm/sec CNT100;
   1:  PR[91] = PR[90];
   1:  PR[91,1] = PR[90,1] + -0.525;
   1:  PR[91,2] = PR[90,2] + 23.348;
   1:  PR[91,3] = PR[90,3] + 63.895;
   1:L PR[91] R[100]mm/sec CNT100;
   1:  PR[91,1] = PR[90,1] + -5.615;
   1:  PR[91,2] = PR[90,2] + 23.580;
   1:L PR[91] R[100]mm/sec CNT100;
   1:  PR[91,1] = PR[90,1] + -5.644;
   1:  PR[91,2] = PR[90,2] + 23.578;
   1:L PR[91] R[100]mm/sec CNT100;
   1:  PR[91,1] = PR[90,1] + -10.891;
   1:  PR[91,2] = PR[90,2] + 22.692;
   1:L PR[91] R[100]mm/sec CNT100;
   1:  PR[91,1] = PR[90,1] + -15.791;
   1:  PR[91,2] = PR[90,2] + 20.725;
   1:L PR[91] R[100]mm/sec CNT100;
   1:  PR[91,1] = PR[90,1] + -20.159;
   1:  PR[91,2] = PR[90,2] + 17.777;
   1:L PR[91] R[100]mm/sec CNT100;
   1:  PR[91,1] = PR[90,1] + -23.779;
   1:  PR[91,2] = PR[90,2] + 13.998;
   1:L PR[91] R[100]mm/sec CNT100;
   1:  PR[91,1] = PR[90,1] + -26.481;
   1:  PR[91,2] = PR[90,2] + 9.560;
   1:L PR[91] R[100]mm/sec CNT100;
   1:  PR[91,1] = PR[90,1] + -28.144;
   1:  PR[91,2] = PR[90,2] + 4.705;
   1:L PR[91] R[100]mm/sec CNT100;
   1:  PR[91,1] = PR[90,1] + -28.220;
   1:  PR[91,2] = PR[90,2] + 3.942;
   1:L PR[91] R[100]mm/sec CNT100;
   1:  PR[91,1] = PR[90,1] + -28.705;
   1:  PR[91,2] = PR[90,2] + -0.466;
   1:L PR[91] R[100]mm/sec CNT100;
   1:  PR[91,1] = PR[90,1] + -28.700;
   1:  PR[91,2] = PR[90,2] + -0.525;
   1:L PR[91] R[100]mm/sec CNT100;
   1:  PR[91,1] = PR[90,1] + -28.148;
   1:  PR[91,2] = PR[90,2] + -5.540;
   1:L PR[91] R[100]mm/sec CNT100;
   1:  PR[91,1] = PR[90,1] + -26.481;
   1:  PR[91,2] = PR[90,2] + -10.407;
   1:L PR[91] R[100]mm/sec CNT100;
   1:  PR[91,1] = PR[90,1] + -23.780;
   1:  PR[91,2] = PR[90,2] + -14.845;
   1:L PR[91] R[100]mm/sec CNT100;
   1:  PR[91,1] = PR[90,1] + -20.160;
   1:  PR[91,2] = PR[90,2] + -18.624;
   1:L PR[91] R[100]mm/sec CNT100;
   1:  PR[91,1] = PR[90,1] + -15.822;
   1:  PR[91,2] = PR[90,2] + -21.555;
   1:L PR[91] R[100]mm/sec CNT100;
   1:  PR[91,1] = PR[90,1] + -10.879;
   1:  PR[91,2] = PR[90,2] + -23.543;
   1:L PR[91] R[100]mm/sec CNT100;
   1:  PR[91,1] = PR[90,1] + -10.865;
   1:  PR[91,2] = PR[90,2] + -23.547;
   1:L PR[91] R[100]mm/sec CNT100;
   1:  PR[91,1] = PR[90,1] + -5.750;
   1:  PR[91,2] = PR[90,2] + -24.409;
   1:L PR[91] R[100]mm/sec CNT100;
   1:  PR[91,1] = PR[90,1] + -5.575;
   1:  PR[91,2] = PR[90,2] + -24.425;
   1:L PR[91] R[100]mm/sec CNT100;
   1:  PR[91,1] = PR[90,1] + -0.525;
   1:  PR[91,2] = PR[90,2] + -24.195;
   1:L PR[91] R[100]mm/sec CNT100;
   1:  PR[91,1] = PR[90,1] + 0.045;
   1:L PR[91] R[100]mm/sec CNT100;
   1:  PR[91,1] = PR[90,1] + 5.089;
   1:  PR[91,2] = PR[90,2] + -24.424;
   1:L PR[91] R[100]mm/sec CNT100;
   1:  PR[91,1] = PR[90,1] + 5.291;
   1:  PR[91,2] = PR[90,2] + -24.406;
   1:L PR[91] R[100]mm/sec CNT100;
   1:  PR[91,1] = PR[90,1] + 10.388;
   1:  PR[91,2] = PR[90,2] + -23.546;
   1:L PR[91] R[100]mm/sec CNT100;
   1:  PR[91,1] = PR[90,1] + 10.406;
   1:  PR[91,2] = PR[90,2] + -23.541;
   1:L PR[91] R[100]mm/sec CNT100;
   1:  PR[91,1] = PR[90,1] + 15.348;
   1:  PR[91,2] = PR[90,2] + -21.552;
   1:L PR[91] R[100]mm/sec CNT100;
   1:  PR[91,1] = PR[90,1] + 19.680;
   1:  PR[91,2] = PR[90,2] + -18.624;
   1:L PR[91] R[100]mm/sec CNT100;
   1:  PR[91,1] = PR[90,1] + 23.301;
   1:  PR[91,2] = PR[90,2] + -14.843;
   1:L PR[91] R[100]mm/sec CNT100;
   1:  PR[91,1] = PR[90,1] + 26.002;
   1:  PR[91,2] = PR[90,2] + -10.406;
   1:L PR[91] R[100]mm/sec CNT100;
   1:  PR[91,1] = PR[90,1] + 27.667;
   1:  PR[91,2] = PR[90,2] + -5.546;
   1:L PR[91] R[100]mm/sec CNT100;
   1:  PR[91,1] = PR[90,1] + 28.225;
   1:  PR[91,2] = PR[90,2] + -0.383;
   1:L PR[91] R[100]mm/sec CNT100;
   1:  PR[91,1] = PR[90,1] + 28.221;
   1:  PR[91,2] = PR[90,2] + -0.321;
   1:L PR[91] R[100]mm/sec CNT100;
   1:  PR[91,1] = PR[90,1] + 27.668;
   1:  PR[91,2] = PR[90,2] + 4.697;
   1:L PR[91] R[100]mm/sec CNT100;
   1:  PR[91,1] = PR[90,1] + 26.001;
   1:  PR[91,2] = PR[90,2] + 9.560;
   1:L PR[91] R[100]mm/sec CNT100;
   1:  PR[91,1] = PR[90,1] + 23.300;
   1:  PR[91,2] = PR[90,2] + 13.997;
   1:L PR[91] R[100]mm/sec CNT100;
   1:  PR[91,1] = PR[90,1] + 19.679;
   1:  PR[91,2] = PR[90,2] + 17.778;
   1:L PR[91] R[100]mm/sec CNT100;
   1:  PR[91,1] = PR[90,1] + 15.312;
   1:  PR[91,2] = PR[90,2] + 20.725;
   1:L PR[91] R[100]mm/sec CNT100;
   1:  PR[91,1] = PR[90,1] + 10.412;
   1:  PR[91,2] = PR[90,2] + 22.691;
   1:L PR[91] R[100]mm/sec CNT100;
   1:  PR[91,1] = PR[90,1] + 5.165;
   1:  PR[91,2] = PR[90,2] + 23.578;
   1:L PR[91] R[100]mm/sec CNT100;
   1:  PR[91,1] = PR[90,1] + 5.136;
   1:  PR[91,2] = PR[90,2] + 23.580;
   1:L PR[91] R[100]mm/sec CNT100;
   1:  PR[91,1] = PR[90,1] + 0.045;
   1:  PR[91,2] = PR[90,2] + 23.348;
   1:L PR[91] R[100]mm/sec CNT100;
   1:  PR[91] = PR[90];
   1:  PR[91,1] = PR[90,1] + -0.488;
   1:  PR[91,2] = PR[90,2] + 23.688;
   1:  PR[91,3] = PR[90,3] + 65.195;
   1:L PR[91] R[100]mm/sec CNT100;
   1:  PR[91,1] = PR[90,1] + -4.976;
   1:  PR[91,2] = PR[90,2] + 23.886;
   1:L PR[91] R[100]mm/sec CNT100;
   1:  PR[91,1] = PR[90,1] + -5.395;
   1:  PR[91,2] = PR[90,2] + 23.860;
   1:L PR[91] R[100]mm/sec CNT100;
   1:  PR[91,1] = PR[90,1] + -9.997;
   1:  PR[91,2] = PR[90,2] + 23.086;
   1:L PR[91] R[100]mm/sec CNT100;
   1:  PR[91,1] = PR[90,1] + -10.404;
   1:  PR[91,2] = PR[90,2] + 23.010;
   1:L PR[91] R[100]mm/sec CNT100;
   1:  PR[91,1] = PR[90,1] + -10.735;
   1:  PR[91,2] = PR[90,2] + 22.904;
   1:L PR[91] R[100]mm/sec CNT100;
   1:  PR[91,1] = PR[90,1] + -15.175;
   1:  PR[91,2] = PR[90,2] + 21.126;
   1:L PR[91] R[100]mm/sec CNT100;
   1:  PR[91,1] = PR[90,1] + -15.391;
   1:  PR[91,2] = PR[90,2] + 21.027;
   1:L PR[91] R[100]mm/sec CNT100;
   1:  PR[91,1] = PR[90,1] + -19.510;
   1:  PR[91,2] = PR[90,2] + 18.244;
   1:L PR[91] R[100]mm/sec CNT100;
   1:  PR[91,1] = PR[90,1] + -19.773;
   1:  PR[91,2] = PR[90,2] + 18.082;
   1:L PR[91] R[100]mm/sec CNT100;
   1:  PR[91,1] = PR[90,1] + -19.853;
   1:  PR[91,2] = PR[90,2] + 18.017;
   1:L PR[91] R[100]mm/sec CNT100;
   1:  PR[91,1] = PR[90,1] + -23.303;
   1:  PR[91,2] = PR[90,2] + 14.397;
   1:L PR[91] R[100]mm/sec CNT100;
   1:  PR[91,1] = PR[90,1] + -23.500;
   1:  PR[91,2] = PR[90,2] + 14.177;
   1:L PR[91] R[100]mm/sec CNT100;
   1:  PR[91,1] = PR[90,1] + -26.213;
   1:  PR[91,2] = PR[90,2] + 9.688;
   1:L PR[91] R[100]mm/sec CNT100;
   1:  PR[91,1] = PR[90,1] + -27.896;
   1:  PR[91,2] = PR[90,2] + 4.782;
   1:L PR[91] R[100]mm/sec CNT100;
   1:  PR[91,1] = PR[90,1] + -27.900;
   1:  PR[91,2] = PR[90,2] + 4.769;
   1:L PR[91] R[100]mm/sec CNT100;
   1:  PR[91,1] = PR[90,1] + -27.903;
   1:  PR[91,2] = PR[90,2] + 4.749;
   1:L PR[91] R[100]mm/sec CNT100;
   1:  PR[91,1] = PR[90,1] + -28.464;
   1:  PR[91,2] = PR[90,2] + -0.374;
   1:L PR[91] R[100]mm/sec CNT100;
   1:  PR[91,1] = PR[90,1] + -27.894;
   1:  PR[91,2] = PR[90,2] + -5.590;
   1:L PR[91] R[100]mm/sec CNT100;
   1:  PR[91,1] = PR[90,1] + -26.218;
   1:  PR[91,2] = PR[90,2] + -10.531;
   1:L PR[91] R[100]mm/sec CNT100;
   1:  PR[91,1] = PR[90,1] + -26.119;
   1:  PR[91,2] = PR[90,2] + -10.708;
   1:L PR[91] R[100]mm/sec CNT100;
   1:  PR[91,1] = PR[90,1] + -23.485;
   1:  PR[91,2] = PR[90,2] + -15.054;
   1:L PR[91] R[100]mm/sec CNT100;
   1:  PR[91,1] = PR[90,1] + -23.465;
   1:  PR[91,2] = PR[90,2] + -15.080;
   1:L PR[91] R[100]mm/sec CNT100;
   1:  PR[91,1] = PR[90,1] + -19.885;
   1:  PR[91,2] = PR[90,2] + -18.831;
   1:L PR[91] R[100]mm/sec CNT100;
   1:  PR[91,1] = PR[90,1] + -19.569;
   1:  PR[91,2] = PR[90,2] + -19.067;
   1:L PR[91] R[100]mm/sec CNT100;
   1:  PR[91,1] = PR[90,1] + -15.552;
   1:  PR[91,2] = PR[90,2] + -21.784;
   1:L PR[91] R[100]mm/sec CNT100;
   1:  PR[91,1] = PR[90,1] + -15.109;
   1:  PR[91,2] = PR[90,2] + -21.999;
   1:L PR[91] R[100]mm/sec CNT100;
   1:  PR[91,1] = PR[90,1] + -10.742;
   1:  PR[91,2] = PR[90,2] + -23.748;
   1:L PR[91] R[100]mm/sec CNT100;
   1:  PR[91,1] = PR[90,1] + -10.148;
   1:  PR[91,2] = PR[90,2] + -23.911;
   1:L PR[91] R[100]mm/sec CNT100;
   1:  PR[91,1] = PR[90,1] + -5.679;
   1:  PR[91,2] = PR[90,2] + -24.665;
   1:L PR[91] R[100]mm/sec CNT100;
   1:  PR[91,1] = PR[90,1] + -4.916;
   1:  PR[91,2] = PR[90,2] + -24.731;
   1:L PR[91] R[100]mm/sec CNT100;
   1:  PR[91,1] = PR[90,1] + -0.495;
   1:  PR[91,2] = PR[90,2] + -24.535;
   1:L PR[91] R[100]mm/sec CNT100;
   1:  PR[91,1] = PR[90,1] + 0.015;
   1:L PR[91] R[100]mm/sec CNT100;
   1:  PR[91,1] = PR[90,1] + 4.430;
   1:  PR[91,2] = PR[90,2] + -24.730;
   1:L PR[91] R[100]mm/sec CNT100;
   1:  PR[91,1] = PR[90,1] + 5.258;
   1:  PR[91,2] = PR[90,2] + -24.654;
   1:L PR[91] R[100]mm/sec CNT100;
   1:  PR[91,1] = PR[90,1] + 9.710;
   1:  PR[91,2] = PR[90,2] + -23.903;
   1:L PR[91] R[100]mm/sec CNT100;
   1:  PR[91,1] = PR[90,1] + 10.316;
   1:  PR[91,2] = PR[90,2] + -23.728;
   1:L PR[91] R[100]mm/sec CNT100;
   1:  PR[91,1] = PR[90,1] + 14.674;
   1:  PR[91,2] = PR[90,2] + -21.982;
   1:L PR[91] R[100]mm/sec CNT100;
   1:  PR[91,1] = PR[90,1] + 15.094;
   1:  PR[91,2] = PR[90,2] + -21.772;
   1:L PR[91] R[100]mm/sec CNT100;
   1:  PR[91,1] = PR[90,1] + 19.113;
   1:  PR[91,2] = PR[90,2] + -19.053;
   1:L PR[91] R[100]mm/sec CNT100;
   1:  PR[91,1] = PR[90,1] + 19.401;
   1:  PR[91,2] = PR[90,2] + -18.836;
   1:L PR[91] R[100]mm/sec CNT100;
   1:  PR[91,1] = PR[90,1] + 22.825;
   1:  PR[91,2] = PR[90,2] + -15.241;
   1:L PR[91] R[100]mm/sec CNT100;
   1:  PR[91,1] = PR[90,1] + 23.021;
   1:  PR[91,2] = PR[90,2] + -15.021;
   1:L PR[91] R[100]mm/sec CNT100;
   1:  PR[91,1] = PR[90,1] + 25.734;
   1:  PR[91,2] = PR[90,2] + -10.533;
   1:L PR[91] R[100]mm/sec CNT100;
   1:  PR[91,1] = PR[90,1] + 27.416;
   1:  PR[91,2] = PR[90,2] + -5.631;
   1:L PR[91] R[100]mm/sec CNT100;
   1:  PR[91,1] = PR[90,1] + 27.420;
   1:  PR[91,2] = PR[90,2] + -5.618;
   1:L PR[91] R[100]mm/sec CNT100;
   1:  PR[91,1] = PR[90,1] + 27.423;
   1:  PR[91,2] = PR[90,2] + -5.599;
   1:L PR[91] R[100]mm/sec CNT100;
   1:  PR[91,1] = PR[90,1] + 27.984;
   1:  PR[91,2] = PR[90,2] + -0.473;
   1:L PR[91] R[100]mm/sec CNT100;
   1:  PR[91,1] = PR[90,1] + 27.414;
   1:  PR[91,2] = PR[90,2] + 4.746;
   1:L PR[91] R[100]mm/sec CNT100;
   1:  PR[91,1] = PR[90,1] + 25.738;
   1:  PR[91,2] = PR[90,2] + 9.684;
   1:L PR[91] R[100]mm/sec CNT100;
   1:  PR[91,1] = PR[90,1] + 25.639;
   1:  PR[91,2] = PR[90,2] + 9.861;
   1:L PR[91] R[100]mm/sec CNT100;
   1:  PR[91,1] = PR[90,1] + 23.005;
   1:  PR[91,2] = PR[90,2] + 14.207;
   1:L PR[91] R[100]mm/sec CNT100;
   1:  PR[91,1] = PR[90,1] + 22.984;
   1:  PR[91,2] = PR[90,2] + 14.233;
   1:L PR[91] R[100]mm/sec CNT100;
   1:  PR[91,1] = PR[90,1] + 19.374;
   1:  PR[91,2] = PR[90,2] + 18.017;
   1:L PR[91] R[100]mm/sec CNT100;
   1:  PR[91,1] = PR[90,1] + 19.256;
   1:  PR[91,2] = PR[90,2] + 18.113;
   1:L PR[91] R[100]mm/sec CNT100;
   1:  PR[91,1] = PR[90,1] + 15.208;
   1:  PR[91,2] = PR[90,2] + 20.850;
   1:L PR[91] R[100]mm/sec CNT100;
   1:  PR[91,1] = PR[90,1] + 14.955;
   1:  PR[91,2] = PR[90,2] + 21.007;
   1:L PR[91] R[100]mm/sec CNT100;
   1:  PR[91,1] = PR[90,1] + 14.696;
   1:  PR[91,2] = PR[90,2] + 21.126;
   1:L PR[91] R[100]mm/sec CNT100;
   1:  PR[91,1] = PR[90,1] + 10.256;
   1:  PR[91,2] = PR[90,2] + 22.904;
   1:L PR[91] R[100]mm/sec CNT100;
   1:  PR[91,1] = PR[90,1] + 9.946;
   1:  PR[91,2] = PR[90,2] + 23.003;
   1:L PR[91] R[100]mm/sec CNT100;
   1:  PR[91,1] = PR[90,1] + 5.432;
   1:  PR[91,2] = PR[90,2] + 23.761;
   1:L PR[91] R[100]mm/sec CNT100;
   1:  PR[91,1] = PR[90,1] + 4.894;
   1:  PR[91,2] = PR[90,2] + 23.862;
   1:L PR[91] R[100]mm/sec CNT100;
   1:  PR[91,1] = PR[90,1] + 4.496;
   1:  PR[91,2] = PR[90,2] + 23.886;
   1:L PR[91] R[100]mm/sec CNT100;
   1:  PR[91,1] = PR[90,1] + 0.015;
   1:  PR[91,2] = PR[90,2] + 23.688;
   1:L PR[91] R[100]mm/sec CNT100;
   1:  PR[91] = PR[90];
   1:  PR[91,1] = PR[90,1] + -0.466;
   1:  PR[91,2] = PR[90,2] + 24.024;
   1:  PR[91,3] = PR[90,3] + 66.495;
   1:L PR[91] R[100]mm/sec CNT100;
   1:  PR[91,1] = PR[90,1] + -4.337;
   1:  PR[91,2] = PR[90,2] + 24.193;
   1:L PR[91] R[100]mm/sec CNT100;
   1:  PR[91,1] = PR[90,1] + -5.145;
   1:  PR[91,2] = PR[90,2] + 24.143;
   1:L PR[91] R[100]mm/sec CNT100;
   1:  PR[91,1] = PR[90,1] + -9.111;
   1:  PR[91,2] = PR[90,2] + 23.476;
   1:L PR[91] R[100]mm/sec CNT100;
   1:  PR[91,1] = PR[90,1] + -9.911;
   1:  PR[91,2] = PR[90,2] + 23.326;
   1:L PR[91] R[100]mm/sec CNT100;
   1:  PR[91,1] = PR[90,1] + -10.624;
   1:  PR[91,2] = PR[90,2] + 23.099;
   1:L PR[91] R[100]mm/sec CNT100;
   1:  PR[91,1] = PR[90,1] + -14.451;
   1:  PR[91,2] = PR[90,2] + 21.567;
   1:L PR[91] R[100]mm/sec CNT100;
   1:  PR[91,1] = PR[90,1] + -15.041;
   1:  PR[91,2] = PR[90,2] + 21.295;
   1:L PR[91] R[100]mm/sec CNT100;
   1:  PR[91,1] = PR[90,1] + -18.591;
   1:  PR[91,2] = PR[90,2] + 18.897;
   1:L PR[91] R[100]mm/sec CNT100;
   1:  PR[91,1] = PR[90,1] + -19.214;
   1:  PR[91,2] = PR[90,2] + 18.511;
   1:L PR[91] R[100]mm/sec CNT100;
   1:  PR[91,1] = PR[90,1] + -19.625;
   1:  PR[91,2] = PR[90,2] + 18.181;
   1:L PR[91] R[100]mm/sec CNT100;
   1:  PR[91,1] = PR[90,1] + -22.594;
   1:  PR[91,2] = PR[90,2] + 15.065;
   1:L PR[91] R[100]mm/sec CNT100;
   1:  PR[91,1] = PR[90,1] + -23.272;
   1:  PR[91,2] = PR[90,2] + 14.306;
   1:L PR[91] R[100]mm/sec CNT100;
   1:  PR[91,1] = PR[90,1] + -25.512;
   1:  PR[91,2] = PR[90,2] + 10.610;
   1:L PR[91] R[100]mm/sec CNT100;
   1:  PR[91,1] = PR[90,1] + -25.964;
   1:  PR[91,2] = PR[90,2] + 9.834;
   1:L PR[91] R[100]mm/sec CNT100;
   1:  PR[91,1] = PR[90,1] + -27.386;
   1:  PR[91,2] = PR[90,2] + 5.665;
   1:L PR[91] R[100]mm/sec CNT100;
   1:  PR[91,1] = PR[90,1] + -27.576;
   1:  PR[91,2] = PR[90,2] + 5.188;
   1:L PR[91] R[100]mm/sec CNT100;
   1:  PR[91,1] = PR[90,1] + -27.670;
   1:  PR[91,2] = PR[90,2] + 4.853;
   1:L PR[91] R[100]mm/sec CNT100;
   1:  PR[91,1] = PR[90,1] + -27.740;
   1:  PR[91,2] = PR[90,2] + 4.436;
   1:L PR[91] R[100]mm/sec CNT100;
   1:  PR[91,1] = PR[90,1] + -28.226;
   1:  PR[91,2] = PR[90,2] + -0.007;
   1:L PR[91] R[100]mm/sec CNT100;
   1:  PR[91,1] = PR[90,1] + -28.246;
   1:  PR[91,2] = PR[90,2] + -0.361;
   1:L PR[91] R[100]mm/sec CNT100;
   1:  PR[91,1] = PR[90,1] + -27.672;
   1:  PR[91,2] = PR[90,2] + -5.649;
   1:L PR[91] R[100]mm/sec CNT100;
   1:  PR[91,1] = PR[90,1] + -27.408;
   1:  PR[91,2] = PR[90,2] + -6.482;
   1:L PR[91] R[100]mm/sec CNT100;
   1:  PR[91,1] = PR[90,1] + -26.009;
   1:  PR[91,2] = PR[90,2] + -10.584;
   1:L PR[91] R[100]mm/sec CNT100;
   1:  PR[91,1] = PR[90,1] + -25.550;
   1:  PR[91,2] = PR[90,2] + -11.406;
   1:L PR[91] R[100]mm/sec CNT100;
   1:  PR[91,1] = PR[90,1] + -23.286;
   1:  PR[91,2] = PR[90,2] + -15.143;
   1:L PR[91] R[100]mm/sec CNT100;
   1:  PR[91,1] = PR[90,1] + -23.031;
   1:  PR[91,2] = PR[90,2] + -15.467;
   1:L PR[91] R[100]mm/sec CNT100;
   1:  PR[91,1] = PR[90,1] + -19.658;
   1:  PR[91,2] = PR[90,2] + -18.994;
   1:L PR[91] R[100]mm/sec CNT100;
   1:  PR[91,1] = PR[90,1] + -18.800;
   1:  PR[91,2] = PR[90,2] + -19.634;
   1:L PR[91] R[100]mm/sec CNT100;
   1:  PR[91,1] = PR[90,1] + -15.353;
   1:  PR[91,2] = PR[90,2] + -21.966;
   1:L PR[91] R[100]mm/sec CNT100;
   1:  PR[91,1] = PR[90,1] + -14.346;
   1:  PR[91,2] = PR[90,2] + -22.454;
   1:L PR[91] R[100]mm/sec CNT100;
   1:  PR[91,1] = PR[90,1] + -10.604;
   1:  PR[91,2] = PR[90,2] + -23.953;
   1:L PR[91] R[100]mm/sec CNT100;
   1:  PR[91,1] = PR[90,1] + -9.431;
   1:  PR[91,2] = PR[90,2] + -24.275;
   1:L PR[91] R[100]mm/sec CNT100;
   1:  PR[91,1] = PR[90,1] + -5.608;
   1:  PR[91,2] = PR[90,2] + -24.920;
   1:L PR[91] R[100]mm/sec CNT100;
   1:  PR[91,1] = PR[90,1] + -4.259;
   1:  PR[91,2] = PR[90,2] + -25.037;
   1:L PR[91] R[100]mm/sec CNT100;
   1:  PR[91,1] = PR[90,1] + -0.466;
   1:  PR[91,2] = PR[90,2] + -24.871;
   1:L PR[91] R[100]mm/sec CNT100;
   1:  PR[91,1] = PR[90,1] + -0.014;
   1:L PR[91] R[100]mm/sec CNT100;
   1:  PR[91,1] = PR[90,1] + 3.773;
   1:  PR[91,2] = PR[90,2] + -25.036;
   1:L PR[91] R[100]mm/sec CNT100;
   1:  PR[91,1] = PR[90,1] + 5.224;
   1:  PR[91,2] = PR[90,2] + -24.902;
   1:L PR[91] R[100]mm/sec CNT100;
   1:  PR[91,1] = PR[90,1] + 9.032;
   1:  PR[91,2] = PR[90,2] + -24.260;
   1:L PR[91] R[100]mm/sec CNT100;
   1:  PR[91,1] = PR[90,1] + 10.223;
   1:  PR[91,2] = PR[90,2] + -23.915;
   1:L PR[91] R[100]mm/sec CNT100;
   1:  PR[91,1] = PR[90,1] + 13.959;
   1:  PR[91,2] = PR[90,2] + -22.418;
   1:L PR[91] R[100]mm/sec CNT100;
   1:  PR[91,1] = PR[90,1] + 14.921;
   1:  PR[91,2] = PR[90,2] + -21.937;
   1:L PR[91] R[100]mm/sec CNT100;
   1:  PR[91,1] = PR[90,1] + 18.372;
   1:  PR[91,2] = PR[90,2] + -19.603;
   1:L PR[91] R[100]mm/sec CNT100;
   1:  PR[91,1] = PR[90,1] + 19.173;
   1:  PR[91,2] = PR[90,2] + -18.999;
   1:L PR[91] R[100]mm/sec CNT100;
   1:  PR[91,1] = PR[90,1] + 22.116;
   1:  PR[91,2] = PR[90,2] + -15.909;
   1:L PR[91] R[100]mm/sec CNT100;
   1:  PR[91,1] = PR[90,1] + 22.793;
   1:  PR[91,2] = PR[90,2] + -15.150;
   1:L PR[91] R[100]mm/sec CNT100;
   1:  PR[91,1] = PR[90,1] + 25.033;
   1:  PR[91,2] = PR[90,2] + -11.455;
   1:L PR[91] R[100]mm/sec CNT100;
   1:  PR[91,1] = PR[90,1] + 25.485;
   1:  PR[91,2] = PR[90,2] + -10.680;
   1:L PR[91] R[100]mm/sec CNT100;
   1:  PR[91,1] = PR[90,1] + 26.907;
   1:  PR[91,2] = PR[90,2] + -6.514;
   1:L PR[91] R[100]mm/sec CNT100;
   1:  PR[91,1] = PR[90,1] + 27.096;
   1:  PR[91,2] = PR[90,2] + -6.037;
   1:L PR[91] R[100]mm/sec CNT100;
   1:  PR[91,1] = PR[90,1] + 27.190;
   1:  PR[91,2] = PR[90,2] + -5.702;
   1:L PR[91] R[100]mm/sec CNT100;
   1:  PR[91,1] = PR[90,1] + 27.260;
   1:  PR[91,2] = PR[90,2] + -5.285;
   1:L PR[91] R[100]mm/sec CNT100;
   1:  PR[91,1] = PR[90,1] + 27.746;
   1:  PR[91,2] = PR[90,2] + -0.840;
   1:L PR[91] R[100]mm/sec CNT100;
   1:  PR[91,1] = PR[90,1] + 27.766;
   1:  PR[91,2] = PR[90,2] + -0.487;
   1:L PR[91] R[100]mm/sec CNT100;
   1:  PR[91,1] = PR[90,1] + 27.193;
   1:  PR[91,2] = PR[90,2] + 4.804;
   1:L PR[91] R[100]mm/sec CNT100;
   1:  PR[91,1] = PR[90,1] + 26.929;
   1:  PR[91,2] = PR[90,2] + 5.637;
   1:L PR[91] R[100]mm/sec CNT100;
   1:  PR[91,1] = PR[90,1] + 25.530;
   1:  PR[91,2] = PR[90,2] + 9.737;
   1:L PR[91] R[100]mm/sec CNT100;
   1:  PR[91,1] = PR[90,1] + 25.070;
   1:  PR[91,2] = PR[90,2] + 10.559;
   1:L PR[91] R[100]mm/sec CNT100;
   1:  PR[91,1] = PR[90,1] + 22.805;
   1:  PR[91,2] = PR[90,2] + 14.296;
   1:L PR[91] R[100]mm/sec CNT100;
   1:  PR[91,1] = PR[90,1] + 22.550;
   1:  PR[91,2] = PR[90,2] + 14.620;
   1:L PR[91] R[100]mm/sec CNT100;
   1:  PR[91,1] = PR[90,1] + 19.147;
   1:  PR[91,2] = PR[90,2] + 18.179;
   1:L PR[91] R[100]mm/sec CNT100;
   1:  PR[91,1] = PR[90,1] + 18.697;
   1:  PR[91,2] = PR[90,2] + 18.541;
   1:L PR[91] R[100]mm/sec CNT100;
   1:  PR[91,1] = PR[90,1] + 15.209;
   1:  PR[91,2] = PR[90,2] + 20.901;
   1:L PR[91] R[100]mm/sec CNT100;
   1:  PR[91,1] = PR[90,1] + 14.605;
   1:  PR[91,2] = PR[90,2] + 21.275;
   1:L PR[91] R[100]mm/sec CNT100;
   1:  PR[91,1] = PR[90,1] + 13.971;
   1:  PR[91,2] = PR[90,2] + 21.567;
   1:L PR[91] R[100]mm/sec CNT100;
   1:  PR[91,1] = PR[90,1] + 10.145;
   1:  PR[91,2] = PR[90,2] + 23.099;
   1:L PR[91] R[100]mm/sec CNT100;
   1:  PR[91,1] = PR[90,1] + 9.453;
   1:  PR[91,2] = PR[90,2] + 23.319;
   1:L PR[91] R[100]mm/sec CNT100;
   1:  PR[91,1] = PR[90,1] + 5.564;
   1:  PR[91,2] = PR[90,2] + 23.972;
   1:L PR[91] R[100]mm/sec CNT100;
   1:  PR[91,1] = PR[90,1] + 4.644;
   1:  PR[91,2] = PR[90,2] + 24.144;
   1:L PR[91] R[100]mm/sec CNT100;
   1:  PR[91,1] = PR[90,1] + 3.857;
   1:  PR[91,2] = PR[90,2] + 24.193;
   1:L PR[91] R[100]mm/sec CNT100;
   1:  PR[91,1] = PR[90,1] + -0.014;
   1:  PR[91,2] = PR[90,2] + 24.024;
   1:L PR[91] R[100]mm/sec CNT100;
   1:  PR[91] = PR[90];
   1:  PR[91,1] = PR[90,1] + -0.437;
   1:  PR[91,2] = PR[90,2] + 24.360;
   1:  PR[91,3] = PR[90,3] + 67.795;
   1:L PR[91] R[100]mm/sec CNT100;
   1:  PR[91,1] = PR[90,1] + -3.699;
   1:  PR[91,2] = PR[90,2] + 24.500;
   1:L PR[91] R[100]mm/sec CNT100;
   1:  PR[91,1] = PR[90,1] + -4.895;
   1:  PR[91,2] = PR[90,2] + 24.426;
   1:L PR[91] R[100]mm/sec CNT100;
   1:  PR[91,1] = PR[90,1] + -8.225;
   1:  PR[91,2] = PR[90,2] + 23.865;
   1:L PR[91] R[100]mm/sec CNT100;
   1:  PR[91,1] = PR[90,1] + -9.418;
   1:  PR[91,2] = PR[90,2] + 23.642;
   1:L PR[91] R[100]mm/sec CNT100;
   1:  PR[91,1] = PR[90,1] + -10.513;
   1:  PR[91,2] = PR[90,2] + 23.294;
   1:L PR[91] R[100]mm/sec CNT100;
   1:  PR[91,1] = PR[90,1] + -13.726;
   1:  PR[91,2] = PR[90,2] + 22.007;
   1:L PR[91] R[100]mm/sec CNT100;
   1:  PR[91,1] = PR[90,1] + -14.691;
   1:  PR[91,2] = PR[90,2] + 21.563;
   1:L PR[91] R[100]mm/sec CNT100;
   1:  PR[91,1] = PR[90,1] + -17.673;
   1:  PR[91,2] = PR[90,2] + 19.549;
   1:L PR[91] R[100]mm/sec CNT100;
   1:  PR[91,1] = PR[90,1] + -18.656;
   1:  PR[91,2] = PR[90,2] + 18.940;
   1:L PR[91] R[100]mm/sec CNT100;
   1:  PR[91,1] = PR[90,1] + -19.397;
   1:  PR[91,2] = PR[90,2] + 18.344;
   1:L PR[91] R[100]mm/sec CNT100;
   1:  PR[91,1] = PR[90,1] + -21.885;
   1:  PR[91,2] = PR[90,2] + 15.733;
   1:L PR[91] R[100]mm/sec CNT100;
   1:  PR[91,1] = PR[90,1] + -23.042;
   1:  PR[91,2] = PR[90,2] + 14.436;
   1:L PR[91] R[100]mm/sec CNT100;
   1:  PR[91,1] = PR[90,1] + -24.913;
   1:  PR[91,2] = PR[90,2] + 11.351;
   1:L PR[91] R[100]mm/sec CNT100;
   1:  PR[91,1] = PR[90,1] + -25.723;
   1:  PR[91,2] = PR[90,2] + 9.962;
   1:L PR[91] R[100]mm/sec CNT100;
   1:  PR[91,1] = PR[90,1] + -26.912;
   1:  PR[91,2] = PR[90,2] + 6.476;
   1:L PR[91] R[100]mm/sec CNT100;
   1:  PR[91,1] = PR[90,1] + -27.240;
   1:  PR[91,2] = PR[90,2] + 5.650;
   1:L PR[91] R[100]mm/sec CNT100;
   1:  PR[91,1] = PR[90,1] + -27.440;
   1:  PR[91,2] = PR[90,2] + 4.938;
   1:L PR[91] R[100]mm/sec CNT100;
   1:  PR[91,1] = PR[90,1] + -27.576;
   1:  PR[91,2] = PR[90,2] + 4.123;
   1:L PR[91] R[100]mm/sec CNT100;
   1:  PR[91,1] = PR[90,1] + -27.983;
   1:  PR[91,2] = PR[90,2] + 0.406;
   1:L PR[91] R[100]mm/sec CNT100;
   1:  PR[91,1] = PR[90,1] + -28.026;
   1:  PR[91,2] = PR[90,2] + -0.362;
   1:L PR[91] R[100]mm/sec CNT100;
   1:  PR[91,1] = PR[90,1] + -27.453;
   1:  PR[91,2] = PR[90,2] + -5.684;
   1:L PR[91] R[100]mm/sec CNT100;
   1:  PR[91,1] = PR[90,1] + -26.966;
   1:  PR[91,2] = PR[90,2] + -7.220;
   1:L PR[91] R[100]mm/sec CNT100;
   1:  PR[91,1] = PR[90,1] + -25.800;
   1:  PR[91,2] = PR[90,2] + -10.639;
   1:L PR[91] R[100]mm/sec CNT100;
   1:  PR[91,1] = PR[90,1] + -24.981;
   1:  PR[91,2] = PR[90,2] + -12.105;
   1:L PR[91] R[100]mm/sec CNT100;
   1:  PR[91,1] = PR[90,1] + -23.086;
   1:  PR[91,2] = PR[90,2] + -15.232;
   1:L PR[91] R[100]mm/sec CNT100;
   1:  PR[91,1] = PR[90,1] + -22.595;
   1:  PR[91,2] = PR[90,2] + -15.857;
   1:L PR[91] R[100]mm/sec CNT100;
   1:  PR[91,1] = PR[90,1] + -20.102;
   1:  PR[91,2] = PR[90,2] + -18.475;
   1:L PR[91] R[100]mm/sec CNT100;
   1:  PR[91,1] = PR[90,1] + -19.442;
   1:  PR[91,2] = PR[90,2] + -19.148;
   1:L PR[91] R[100]mm/sec CNT100;
   1:  PR[91,1] = PR[90,1] + -18.031;
   1:  PR[91,2] = PR[90,2] + -20.201;
   1:L PR[91] R[100]mm/sec CNT100;
   1:  PR[91,1] = PR[90,1] + -15.153;
   1:  PR[91,2] = PR[90,2] + -22.148;
   1:L PR[91] R[100]mm/sec CNT100;
   1:  PR[91,1] = PR[90,1] + -13.583;
   1:  PR[91,2] = PR[90,2] + -22.909;
   1:L PR[91] R[100]mm/sec CNT100;
   1:  PR[91,1] = PR[90,1] + -10.465;
   1:  PR[91,2] = PR[90,2] + -24.158;
   1:L PR[91] R[100]mm/sec CNT100;
   1:  PR[91,1] = PR[90,1] + -8.714;
   1:  PR[91,2] = PR[90,2] + -24.639;
   1:L PR[91] R[100]mm/sec CNT100;
   1:  PR[91,1] = PR[90,1] + -5.537;
   1:  PR[91,2] = PR[90,2] + -25.175;
   1:L PR[91] R[100]mm/sec CNT100;
   1:  PR[91,1] = PR[90,1] + -3.601;
   1:  PR[91,2] = PR[90,2] + -25.343;
   1:L PR[91] R[100]mm/sec CNT100;
   1:  PR[91,1] = PR[90,1] + -0.437;
   1:  PR[91,2] = PR[90,2] + -25.207;
   1:L PR[91] R[100]mm/sec CNT100;
   1:  PR[91,1] = PR[90,1] + -0.043;
   1:L PR[91] R[100]mm/sec CNT100;
   1:  PR[91,1] = PR[90,1] + 3.115;
   1:  PR[91,2] = PR[90,2] + -25.342;
   1:L PR[91] R[100]mm/sec CNT100;
   1:  PR[91,1] = PR[90,1] + 5.191;
   1:  PR[91,2] = PR[90,2] + -25.150;
   1:L PR[91] R[100]mm/sec CNT100;
   1:  PR[91,1] = PR[90,1] + 8.354;
   1:  PR[91,2] = PR[90,2] + -24.616;
   1:L PR[91] R[100]mm/sec CNT100;
   1:  PR[91,1] = PR[90,1] + 10.131;
   1:  PR[91,2] = PR[90,2] + -24.102;
   1:L PR[91] R[100]mm/sec CNT100;
   1:  PR[91,1] = PR[90,1] + 13.244;
   1:  PR[91,2] = PR[90,2] + -22.855;
   1:L PR[91] R[100]mm/sec CNT100;
   1:  PR[91,1] = PR[90,1] + 14.749;
   1:  PR[91,2] = PR[90,2] + -22.102;
   1:L PR[91] R[100]mm/sec CNT100;
   1:  PR[91,1] = PR[90,1] + 17.631;
   1:  PR[91,2] = PR[90,2] + -20.153;
   1:L PR[91] R[100]mm/sec CNT100;
   1:  PR[91,1] = PR[90,1] + 18.945;
   1:  PR[91,2] = PR[90,2] + -19.163;
   1:L PR[91] R[100]mm/sec CNT100;
   1:  PR[91,1] = PR[90,1] + 21.406;
   1:  PR[91,2] = PR[90,2] + -16.578;
   1:L PR[91] R[100]mm/sec CNT100;
   1:  PR[91,1] = PR[90,1] + 22.564;
   1:  PR[91,2] = PR[90,2] + -15.281;
   1:L PR[91] R[100]mm/sec CNT100;
   1:  PR[91,1] = PR[90,1] + 24.434;
   1:  PR[91,2] = PR[90,2] + -12.196;
   1:L PR[91] R[100]mm/sec CNT100;
   1:  PR[91,1] = PR[90,1] + 25.244;
   1:  PR[91,2] = PR[90,2] + -10.807;
   1:L PR[91] R[100]mm/sec CNT100;
   1:  PR[91,1] = PR[90,1] + 26.432;
   1:  PR[91,2] = PR[90,2] + -7.324;
   1:L PR[91] R[100]mm/sec CNT100;
   1:  PR[91,1] = PR[90,1] + 26.761;
   1:  PR[91,2] = PR[90,2] + -6.498;
   1:L PR[91] R[100]mm/sec CNT100;
   1:  PR[91,1] = PR[90,1] + 26.961;
   1:  PR[91,2] = PR[90,2] + -5.786;
   1:L PR[91] R[100]mm/sec CNT100;
   1:  PR[91,1] = PR[90,1] + 27.097;
   1:  PR[91,2] = PR[90,2] + -4.972;
   1:L PR[91] R[100]mm/sec CNT100;
   1:  PR[91,1] = PR[90,1] + 27.504;
   1:  PR[91,2] = PR[90,2] + -1.253;
   1:L PR[91] R[100]mm/sec CNT100;
   1:  PR[91,1] = PR[90,1] + 27.546;
   1:  PR[91,2] = PR[90,2] + -0.486;
   1:L PR[91] R[100]mm/sec CNT100;
   1:  PR[91,1] = PR[90,1] + 26.974;
   1:  PR[91,2] = PR[90,2] + 4.838;
   1:L PR[91] R[100]mm/sec CNT100;
   1:  PR[91,1] = PR[90,1] + 26.487;
   1:  PR[91,2] = PR[90,2] + 6.374;
   1:L PR[91] R[100]mm/sec CNT100;
   1:  PR[91,1] = PR[90,1] + 25.321;
   1:  PR[91,2] = PR[90,2] + 9.792;
   1:L PR[91] R[100]mm/sec CNT100;
   1:  PR[91,1] = PR[90,1] + 24.501;
   1:  PR[91,2] = PR[90,2] + 11.258;
   1:L PR[91] R[100]mm/sec CNT100;
   1:  PR[91,1] = PR[90,1] + 22.605;
   1:  PR[91,2] = PR[90,2] + 14.385;
   1:L PR[91] R[100]mm/sec CNT100;
   1:  PR[91,1] = PR[90,1] + 22.114;
   1:  PR[91,2] = PR[90,2] + 15.010;
   1:L PR[91] R[100]mm/sec CNT100;
   1:  PR[91,1] = PR[90,1] + 19.621;
   1:  PR[91,2] = PR[90,2] + 17.629;
   1:L PR[91] R[100]mm/sec CNT100;
   1:  PR[91,1] = PR[90,1] + 18.931;
   1:  PR[91,2] = PR[90,2] + 18.333;
   1:L PR[91] R[100]mm/sec CNT100;
   1:  PR[91,1] = PR[90,1] + 18.139;
   1:  PR[91,2] = PR[90,2] + 18.970;
   1:L PR[91] R[100]mm/sec CNT100;
   1:  PR[91,1] = PR[90,1] + 15.210;
   1:  PR[91,2] = PR[90,2] + 20.952;
   1:L PR[91] R[100]mm/sec CNT100;
   1:  PR[91,1] = PR[90,1] + 14.255;
   1:  PR[91,2] = PR[90,2] + 21.543;
   1:L PR[91] R[100]mm/sec CNT100;
   1:  PR[91,1] = PR[90,1] + 13.246;
   1:  PR[91,2] = PR[90,2] + 22.007;
   1:L PR[91] R[100]mm/sec CNT100;
   1:  PR[91,1] = PR[90,1] + 10.034;
   1:  PR[91,2] = PR[90,2] + 23.294;
   1:L PR[91] R[100]mm/sec CNT100;
   1:  PR[91,1] = PR[90,1] + 8.960;
   1:  PR[91,2] = PR[90,2] + 23.635;
   1:L PR[91] R[100]mm/sec CNT100;
   1:  PR[91,1] = PR[90,1] + 5.696;
   1:  PR[91,2] = PR[90,2] + 24.184;
   1:L PR[91] R[100]mm/sec CNT100;
   1:  PR[91,1] = PR[90,1] + 4.394;
   1:  PR[91,2] = PR[90,2] + 24.427;
   1:L PR[91] R[100]mm/sec CNT100;
   1:  PR[91,1] = PR[90,1] + 3.219;
   1:  PR[91,2] = PR[90,2] + 24.500;
   1:L PR[91] R[100]mm/sec CNT100;
   1:  PR[91,1] = PR[90,1] + -0.043;
   1:  PR[91,2] = PR[90,2] + 24.360;
   1:L PR[91] R[100]mm/sec CNT100;
   1:  PR[91] = PR[90];
   1:  PR[91,1] = PR[90,1] + -3.056;
   1:  PR[91,2] = PR[90,2] + 24.807;
   1:  PR[91,3] = PR[90,3] + 69.095;
   1:L PR[91] R[100]mm/sec CNT100;
   1:  PR[91,1] = PR[90,1] + -4.646;
   1:  PR[91,2] = PR[90,2] + 24.708;
   1:L PR[91] R[100]mm/sec CNT100;
   1:  PR[91,1] = PR[90,1] + -7.338;
   1:  PR[91,2] = PR[90,2] + 24.255;
   1:L PR[91] R[100]mm/sec CNT100;
   1:  PR[91,1] = PR[90,1] + -8.926;
   1:  PR[91,2] = PR[90,2] + 23.958;
   1:L PR[91] R[100]mm/sec CNT100;
   1:  PR[91,1] = PR[90,1] + -10.402;
   1:  PR[91,2] = PR[90,2] + 23.488;
   1:L PR[91] R[100]mm/sec CNT100;
   1:  PR[91,1] = PR[90,1] + -13.001;
   1:  PR[91,2] = PR[90,2] + 22.448;
   1:L PR[91] R[100]mm/sec CNT100;
   1:  PR[91,1] = PR[90,1] + -14.341;
   1:  PR[91,2] = PR[90,2] + 21.831;
   1:L PR[91] R[100]mm/sec CNT100;
   1:  PR[91,1] = PR[90,1] + -16.754;
   1:  PR[91,2] = PR[90,2] + 20.201;
   1:L PR[91] R[100]mm/sec CNT100;
   1:  PR[91,1] = PR[90,1] + -18.098;
   1:  PR[91,2] = PR[90,2] + 19.369;
   1:L PR[91] R[100]mm/sec CNT100;
   1:  PR[91,1] = PR[90,1] + -19.169;
   1:  PR[91,2] = PR[90,2] + 18.507;
   1:L PR[91] R[100]mm/sec CNT100;
   1:  PR[91,1] = PR[90,1] + -21.176;
   1:  PR[91,2] = PR[90,2] + 16.401;
   1:L PR[91] R[100]mm/sec CNT100;
   1:  PR[91,1] = PR[90,1] + -22.813;
   1:  PR[91,2] = PR[90,2] + 14.566;
   1:L PR[91] R[100]mm/sec CNT100;
   1:  PR[91,1] = PR[90,1] + -24.313;
   1:  PR[91,2] = PR[90,2] + 12.091;
   1:L PR[91] R[100]mm/sec CNT100;
   1:  PR[91,1] = PR[90,1] + -25.481;
   1:  PR[91,2] = PR[90,2] + 10.089;
   1:L PR[91] R[100]mm/sec CNT100;
   1:  PR[91,1] = PR[90,1] + -26.437;
   1:  PR[91,2] = PR[90,2] + 7.287;
   1:L PR[91] R[100]mm/sec CNT100;
   1:  PR[91,1] = PR[90,1] + -26.905;
   1:  PR[91,2] = PR[90,2] + 6.111;
   1:L PR[91] R[100]mm/sec CNT100;
   1:  PR[91,1] = PR[90,1] + -27.210;
   1:  PR[91,2] = PR[90,2] + 5.022;
   1:L PR[91] R[100]mm/sec CNT100;
   1:  PR[91,1] = PR[90,1] + -27.413;
   1:  PR[91,2] = PR[90,2] + 3.810;
   1:L PR[91] R[100]mm/sec CNT100;
   1:  PR[91,1] = PR[90,1] + -27.741;
   1:  PR[91,2] = PR[90,2] + 0.818;
   1:L PR[91] R[100]mm/sec CNT100;
   1:  PR[91,1] = PR[90,1] + -27.806;
   1:  PR[91,2] = PR[90,2] + -0.363;
   1:L PR[91] R[100]mm/sec CNT100;
   1:  PR[91,1] = PR[90,1] + -27.234;
   1:  PR[91,2] = PR[90,2] + -5.718;
   1:L PR[91] R[100]mm/sec CNT100;
   1:  PR[91,1] = PR[90,1] + -26.524;
   1:  PR[91,2] = PR[90,2] + -7.959;
   1:L PR[91] R[100]mm/sec CNT100;
   1:  PR[91,1] = PR[90,1] + -25.591;
   1:  PR[91,2] = PR[90,2] + -10.694;
   1:L PR[91] R[100]mm/sec CNT100;
   1:  PR[91,1] = PR[90,1] + -24.412;
   1:  PR[91,2] = PR[90,2] + -12.803;
   1:L PR[91] R[100]mm/sec CNT100;
   1:  PR[91,1] = PR[90,1] + -22.886;
   1:  PR[91,2] = PR[90,2] + -15.321;
   1:L PR[91] R[100]mm/sec CNT100;
   1:  PR[91,1] = PR[90,1] + -22.160;
   1:  PR[91,2] = PR[90,2] + -16.245;
   1:L PR[91] R[100]mm/sec CNT100;
   1:  PR[91,1] = PR[90,1] + -20.144;
   1:  PR[91,2] = PR[90,2] + -18.362;
   1:L PR[91] R[100]mm/sec CNT100;
   1:  PR[91,1] = PR[90,1] + -19.213;
   1:  PR[91,2] = PR[90,2] + -19.311;
   1:L PR[91] R[100]mm/sec CNT100;
   1:  PR[91,1] = PR[90,1] + -17.262;
   1:  PR[91,2] = PR[90,2] + -20.768;
   1:L PR[91] R[100]mm/sec CNT100;
   1:  PR[91,1] = PR[90,1] + -14.953;
   1:  PR[91,2] = PR[90,2] + -22.330;
   1:L PR[91] R[100]mm/sec CNT100;
   1:  PR[91,1] = PR[90,1] + -12.819;
   1:  PR[91,2] = PR[90,2] + -23.364;
   1:L PR[91] R[100]mm/sec CNT100;
   1:  PR[91,1] = PR[90,1] + -10.326;
   1:  PR[91,2] = PR[90,2] + -24.363;
   1:L PR[91] R[100]mm/sec CNT100;
   1:  PR[91,1] = PR[90,1] + -7.997;
   1:  PR[91,2] = PR[90,2] + -25.003;
   1:L PR[91] R[100]mm/sec CNT100;
   1:  PR[91,1] = PR[90,1] + -5.465;
   1:  PR[91,2] = PR[90,2] + -25.430;
   1:L PR[91] R[100]mm/sec CNT100;
   1:  PR[91,1] = PR[90,1] + -2.939;
   1:  PR[91,2] = PR[90,2] + -25.649;
   1:L PR[91] R[100]mm/sec CNT100;
   1:  PR[91,1] = PR[90,1] + -0.118;
   1:  PR[91,2] = PR[90,2] + -25.541;
   1:L PR[91] R[100]mm/sec CNT100;
   1:  PR[91,1] = PR[90,1] + 2.456;
   1:  PR[91,2] = PR[90,2] + -25.648;
   1:L PR[91] R[100]mm/sec CNT100;
   1:  PR[91,1] = PR[90,1] + 5.158;
   1:  PR[91,2] = PR[90,2] + -25.398;
   1:L PR[91] R[100]mm/sec CNT100;
   1:  PR[91,1] = PR[90,1] + 7.676;
   1:  PR[91,2] = PR[90,2] + -24.973;
   1:L PR[91] R[100]mm/sec CNT100;
   1:  PR[91,1] = PR[90,1] + 10.038;
   1:  PR[91,2] = PR[90,2] + -24.289;
   1:L PR[91] R[100]mm/sec CNT100;
   1:  PR[91,1] = PR[90,1] + 12.528;
   1:  PR[91,2] = PR[90,2] + -23.292;
   1:L PR[91] R[100]mm/sec CNT100;
   1:  PR[91,1] = PR[90,1] + 14.577;
   1:  PR[91,2] = PR[90,2] + -22.268;
   1:L PR[91] R[100]mm/sec CNT100;
   1:  PR[91,1] = PR[90,1] + 16.891;
   1:  PR[91,2] = PR[90,2] + -20.702;
   1:L PR[91] R[100]mm/sec CNT100;
   1:  PR[91,1] = PR[90,1] + 18.716;
   1:  PR[91,2] = PR[90,2] + -19.326;
   1:L PR[91] R[100]mm/sec CNT100;
   1:  PR[91,1] = PR[90,1] + 20.697;
   1:  PR[91,2] = PR[90,2] + -17.246;
   1:L PR[91] R[100]mm/sec CNT100;
   1:  PR[91,1] = PR[90,1] + 22.335;
   1:  PR[91,2] = PR[90,2] + -15.411;
   1:L PR[91] R[100]mm/sec CNT100;
   1:  PR[91,1] = PR[90,1] + 23.835;
   1:  PR[91,2] = PR[90,2] + -12.937;
   1:L PR[91] R[100]mm/sec CNT100;
   1:  PR[91,1] = PR[90,1] + 25.002;
   1:  PR[91,2] = PR[90,2] + -10.934;
   1:L PR[91] R[100]mm/sec CNT100;
   1:  PR[91,1] = PR[90,1] + 25.958;
   1:  PR[91,2] = PR[90,2] + -8.135;
   1:L PR[91] R[100]mm/sec CNT100;
   1:  PR[91,1] = PR[90,1] + 26.425;
   1:  PR[91,2] = PR[90,2] + -6.959;
   1:L PR[91] R[100]mm/sec CNT100;
   1:  PR[91,1] = PR[90,1] + 26.731;
   1:  PR[91,2] = PR[90,2] + -5.870;
   1:L PR[91] R[100]mm/sec CNT100;
   1:  PR[91,1] = PR[90,1] + 26.934;
   1:  PR[91,2] = PR[90,2] + -4.659;
   1:L PR[91] R[100]mm/sec CNT100;
   1:  PR[91,1] = PR[90,1] + 27.261;
   1:  PR[91,2] = PR[90,2] + -1.665;
   1:L PR[91] R[100]mm/sec CNT100;
   1:  PR[91,1] = PR[90,1] + 27.327;
   1:  PR[91,2] = PR[90,2] + -0.485;
   1:L PR[91] R[100]mm/sec CNT100;
   1:  PR[91,1] = PR[90,1] + 26.755;
   1:  PR[91,2] = PR[90,2] + 4.871;
   1:L PR[91] R[100]mm/sec CNT100;
   1:  PR[91,1] = PR[90,1] + 26.044;
   1:  PR[91,2] = PR[90,2] + 7.112;
   1:L PR[91] R[100]mm/sec CNT100;
   1:  PR[91,1] = PR[90,1] + 25.111;
   1:  PR[91,2] = PR[90,2] + 9.847;
   1:L PR[91] R[100]mm/sec CNT100;
   1:  PR[91,1] = PR[90,1] + 23.931;
   1:  PR[91,2] = PR[90,2] + 11.957;
   1:L PR[91] R[100]mm/sec CNT100;
   1:  PR[91,1] = PR[90,1] + 22.406;
   1:  PR[91,2] = PR[90,2] + 14.474;
   1:L PR[91] R[100]mm/sec CNT100;
   1:  PR[91,1] = PR[90,1] + 21.680;
   1:  PR[91,2] = PR[90,2] + 15.398;
   1:L PR[91] R[100]mm/sec CNT100;
   1:  PR[91,1] = PR[90,1] + 19.662;
   1:  PR[91,2] = PR[90,2] + 17.517;
   1:L PR[91] R[100]mm/sec CNT100;
   1:  PR[91,1] = PR[90,1] + 18.703;
   1:  PR[91,2] = PR[90,2] + 18.496;
   1:L PR[91] R[100]mm/sec CNT100;
   1:  PR[91,1] = PR[90,1] + 17.581;
   1:  PR[91,2] = PR[90,2] + 19.399;
   1:L PR[91] R[100]mm/sec CNT100;
   1:  PR[91,1] = PR[90,1] + 15.211;
   1:  PR[91,2] = PR[90,2] + 21.002;
   1:L PR[91] R[100]mm/sec CNT100;
   1:  PR[91,1] = PR[90,1] + 13.905;
   1:  PR[91,2] = PR[90,2] + 21.811;
   1:L PR[91] R[100]mm/sec CNT100;
   1:  PR[91,1] = PR[90,1] + 12.522;
   1:  PR[91,2] = PR[90,2] + 22.448;
   1:L PR[91] R[100]mm/sec CNT100;
   1:  PR[91,1] = PR[90,1] + 9.923;
   1:  PR[91,2] = PR[90,2] + 23.488;
   1:L PR[91] R[100]mm/sec CNT100;
   1:  PR[91,1] = PR[90,1] + 8.467;
   1:  PR[91,2] = PR[90,2] + 23.952;
   1:L PR[91] R[100]mm/sec CNT100;
   1:  PR[91,1] = PR[90,1] + 5.828;
   1:  PR[91,2] = PR[90,2] + 24.395;
   1:L PR[91] R[100]mm/sec CNT100;
   1:  PR[91,1] = PR[90,1] + 4.144;
   1:  PR[91,2] = PR[90,2] + 24.710;
   1:L PR[91] R[100]mm/sec CNT100;
   1:  PR[91,1] = PR[90,1] + 2.579;
   1:  PR[91,2] = PR[90,2] + 24.806;
   1:L PR[91] R[100]mm/sec CNT100;
   1:  PR[91,1] = PR[90,1] + -0.118;
   1:  PR[91,2] = PR[90,2] + 24.693;
   1:L PR[91] R[100]mm/sec CNT100;
   1:  PR[91] = PR[90];
   1:  PR[91,1] = PR[90,1] + -2.417;
   1:  PR[91,2] = PR[90,2] + 25.113;
   1:  PR[91,3] = PR[90,3] + 70.395;
   1:L PR[91] R[100]mm/sec CNT100;
   1:  PR[91,1] = PR[90,1] + -4.396;
   1:  PR[91,2] = PR[90,2] + 24.991;
   1:L PR[91] R[100]mm/sec CNT100;
   1:  PR[91,1] = PR[90,1] + -6.452;
   1:  PR[91,2] = PR[90,2] + 24.645;
   1:L PR[91] R[100]mm/sec CNT100;
   1:  PR[91,1] = PR[90,1] + -8.433;
   1:  PR[91,2] = PR[90,2] + 24.275;
   1:L PR[91] R[100]mm/sec CNT100;
   1:  PR[91,1] = PR[90,1] + -10.291;
   1:  PR[91,2] = PR[90,2] + 23.683;
   1:L PR[91] R[100]mm/sec CNT100;
   1:  PR[91,1] = PR[90,1] + -12.277;
   1:  PR[91,2] = PR[90,2] + 22.888;
   1:L PR[91] R[100]mm/sec CNT100;
   1:  PR[91,1] = PR[90,1] + -13.991;
   1:  PR[91,2] = PR[90,2] + 22.099;
   1:L PR[91] R[100]mm/sec CNT100;
   1:  PR[91,1] = PR[90,1] + -15.835;
   1:  PR[91,2] = PR[90,2] + 20.853;
   1:L PR[91] R[100]mm/sec CNT100;
   1:  PR[91,1] = PR[90,1] + -17.539;
   1:  PR[91,2] = PR[90,2] + 19.798;
   1:L PR[91] R[100]mm/sec CNT100;
   1:  PR[91,1] = PR[90,1] + -18.941;
   1:  PR[91,2] = PR[90,2] + 18.670;
   1:L PR[91] R[100]mm/sec CNT100;
   1:  PR[91,1] = PR[90,1] + -20.467;
   1:  PR[91,2] = PR[90,2] + 17.068;
   1:L PR[91] R[100]mm/sec CNT100;
   1:  PR[91,1] = PR[90,1] + -22.584;
   1:  PR[91,2] = PR[90,2] + 14.697;
   1:L PR[91] R[100]mm/sec CNT100;
   1:  PR[91,1] = PR[90,1] + -23.714;
   1:  PR[91,2] = PR[90,2] + 12.832;
   1:L PR[91] R[100]mm/sec CNT100;
   1:  PR[91,1] = PR[90,1] + -25.240;
   1:  PR[91,2] = PR[90,2] + 10.216;
   1:L PR[91] R[100]mm/sec CNT100;
   1:  PR[91,1] = PR[90,1] + -25.962;
   1:  PR[91,2] = PR[90,2] + 8.098;
   1:L PR[91] R[100]mm/sec CNT100;
   1:  PR[91,1] = PR[90,1] + -26.569;
   1:  PR[91,2] = PR[90,2] + 6.572;
   1:L PR[91] R[100]mm/sec CNT100;
   1:  PR[91,1] = PR[90,1] + -26.980;
   1:  PR[91,2] = PR[90,2] + 5.107;
   1:L PR[91] R[100]mm/sec CNT100;
   1:  PR[91,1] = PR[90,1] + -27.250;
   1:  PR[91,2] = PR[90,2] + 3.497;
   1:L PR[91] R[100]mm/sec CNT100;
   1:  PR[91,1] = PR[90,1] + -27.498;
   1:  PR[91,2] = PR[90,2] + 1.231;
   1:L PR[91] R[100]mm/sec CNT100;
   1:  PR[91,1] = PR[90,1] + -27.587;
   1:  PR[91,2] = PR[90,2] + -0.363;
   1:L PR[91] R[100]mm/sec CNT100;
   1:  PR[91,1] = PR[90,1] + -27.015;
   1:  PR[91,2] = PR[90,2] + -5.753;
   1:L PR[91] R[100]mm/sec CNT100;
   1:  PR[91,1] = PR[90,1] + -26.081;
   1:  PR[91,2] = PR[90,2] + -8.697;
   1:L PR[91] R[100]mm/sec CNT100;
   1:  PR[91,1] = PR[90,1] + -25.382;
   1:  PR[91,2] = PR[90,2] + -10.750;
   1:L PR[91] R[100]mm/sec CNT100;
   1:  PR[91,1] = PR[90,1] + -23.842;
   1:  PR[91,2] = PR[90,2] + -13.502;
   1:L PR[91] R[100]mm/sec CNT100;
   1:  PR[91,1] = PR[90,1] + -22.687;
   1:  PR[91,2] = PR[90,2] + -15.409;
   1:L PR[91] R[100]mm/sec CNT100;
   1:  PR[91,1] = PR[90,1] + -21.726;
   1:  PR[91,2] = PR[90,2] + -16.633;
   1:L PR[91] R[100]mm/sec CNT100;
   1:  PR[91,1] = PR[90,1] + -20.186;
   1:  PR[91,2] = PR[90,2] + -18.249;
   1:L PR[91] R[100]mm/sec CNT100;
   1:  PR[91,1] = PR[90,1] + -18.985;
   1:  PR[91,2] = PR[90,2] + -19.475;
   1:L PR[91] R[100]mm/sec CNT100;
   1:  PR[91,1] = PR[90,1] + -16.493;
   1:  PR[91,2] = PR[90,2] + -21.335;
   1:L PR[91] R[100]mm/sec CNT100;
   1:  PR[91,1] = PR[90,1] + -14.753;
   1:  PR[91,2] = PR[90,2] + -22.512;
   1:L PR[91] R[100]mm/sec CNT100;
   1:  PR[91,1] = PR[90,1] + -12.056;
   1:  PR[91,2] = PR[90,2] + -23.819;
   1:L PR[91] R[100]mm/sec CNT100;
   1:  PR[91,1] = PR[90,1] + -10.187;
   1:  PR[91,2] = PR[90,2] + -24.568;
   1:L PR[91] R[100]mm/sec CNT100;
   1:  PR[91,1] = PR[90,1] + -7.280;
   1:  PR[91,2] = PR[90,2] + -25.367;
   1:L PR[91] R[100]mm/sec CNT100;
   1:  PR[91,1] = PR[90,1] + -5.394;
   1:  PR[91,2] = PR[90,2] + -25.685;
   1:L PR[91] R[100]mm/sec CNT100;
   1:  PR[91,1] = PR[90,1] + -2.281;
   1:  PR[91,2] = PR[90,2] + -25.955;
   1:L PR[91] R[100]mm/sec CNT100;
   1:  PR[91,1] = PR[90,1] + -0.145;
   1:  PR[91,2] = PR[90,2] + -25.874;
   1:L PR[91] R[100]mm/sec CNT100;
   1:  PR[91,1] = PR[90,1] + 1.799;
   1:  PR[91,2] = PR[90,2] + -25.954;
   1:L PR[91] R[100]mm/sec CNT100;
